		Dropoff_Fix08:=80;
		Weld_Fix08:=81;
		Pickup_Fix08:=82;
		Seal_Fix08:=83;
		Stud_Fix08:=84;
		Sweep_Fix08 := 85;

		Dropoff_Fix09:=90;
		Weld_Fix09:=91;
		Pickup_Fix09:=92;
		Seal_Fix09:=93;
		Stud_Fix09:=94;
		Sweep_Fix09 := 95;

		Dropoff_Fix10:=100;
		Weld_Fix10:=101;
		Pickup_Fix10:=102;
		Seal_Fix10:=103;
		Stud_Fix10:=104;
		Sweep_Fix10 := 105;

		Dropoff_Fix11:=110;
		Weld_Fix11:=111;
		Pickup_Fix11:=112;
		Seal_Fix11:=113;
		Stud_Fix11:=114;
		Sweep_Fix11 := 115;

		Dropoff_Fix12:=120;
		Weld_Fix12:=121;
		Pickup_Fix12:=122;
		Seal_Fix12:=123;
		Stud_Fix12:=124;
		Sweep_Fix15 := 125;

		Dropoff_Fix13:=130;
		Weld_Fix13:=131;
		Pickup_Fix13:=132;
		Seal_Fix13:=133;
		Stud_Fix13:=134;
		Sweep_Fix13 := 135;

		Dropoff_Fix14:=140;
		Weld_Fix14:=141;
		Pickup_Fix14:=142;
		Seal_Fix14:=143;
		Stud_Fix14:=144;
		Sweep_Fix14 := 145;

		Dropoff_Fix15:=150;
		Weld_Fix15:=151;
		Pickup_Fix15:=152;
		Seal_Fix15:=153;
		Stud_Fix15:=154;
		Sweep_Fix15 := 155;

		Dropoff_Fix16:=160;
		Weld_Fix16:=161;
		Pickup_Fix16:=162;
		Seal_Fix16:=163;
		Stud_Fix16:=164;
		Sweep_Fix16 := 165;

		(*Tasks Associated with Entire Work Area*)
		Dropoff_Fix101:=200;
		Weld_Fix101:=201;
		Pickup_Fix101:=202;
		Sweep_Fix101:=203;

		Dropoff_Fix102:=204;
		Weld_Fix102:=205;
		Pickup_Fix102:=206;
		Sweep_Fix102:=207;

		Dropoff_Fix103:=208;
		Weld_Fix103:=209;
		Pickup_Fix103:=210;

		Dropoff_Fix104:=212;
		Weld_Fix104:=213;
		Pickup_Fix104:=214;

		Dropoff_Fix105:=216;
		Weld_Fix105:=217;
		Pickup_Fix105:=218;

		Dropoff_Fix106:=220;
		Weld_Fix106:=221;
		Pickup_Fix106:=222;

		Dropoff_Fix107:=224;
		Weld_Fix107:=225;
		Pickup_Fix107:=226;

		Dropoff_Fix108:=228;
		Weld_Fix108:=229;
		Pickup_Fix108:=230;

		Dropoff_Fix109:=232;
		Weld_Fix109:=233;
		Pickup_Fix109:=234;

		Work_Ped01:= 241;
		Work_Ped02:= 242;
		Work_Ped03:= 243;
		Work_Ped04:= 244;
		Work_Ped05:= 245;
		Work_Ped06:= 246;
		Work_Ped07:= 247;
		Work_Ped08:= 248;
		Work_Ped09:= 249;
		Work_Ped10:= 250;
		Work_Ped11:= 251;
		Work_Ped12:= 252;
		Work_Ped13:= 253;
		Work_Ped14:= 254;
		Work_Ped15:= 255;
		Work_Ped16:= 256;
		Work_Ped17:= 257;
		Work_Ped18:= 258;
		Work_Ped19:= 259;
		Work_Ped20:= 260;
		Work_Ped21:= 261;
		Work_Ped22:= 262;
		Work_Ped23:= 263;
		Work_Ped24:= 264;
		Work_Ped25:= 265;
		Work_Ped26:= 266;
		Work_Ped27:= 267;
		Work_Ped28:= 268;
		Work_Ped29:= 269;
		Work_Ped30:= 270;

		Master_Test:= 351;
		Brake_Test:= 352;
		Tip_Dress:=353;
		Tip_Change_EXT:=354;
		Tip_Change:=355;
		Tracc_Tcp:=356;

		(*Robot Types*)
		MOTO_ERC:=1;
		MOTO_MRC:=2;
		MOTO_XRC:=10;
		MOTO_NX100:=20;
		MOTO_DX100:=30;
		MOTO_DX100_Dual:=31;
		MOTO_DX100_32:=40;

		KUKA_KRC2:=51;

		KUKA_KRC4:=60;
		KUKA_KRC4_SAFEOP:=61;
		KUKA_KRC4_SAFEOP_Small:=62;
		KUKA_KRC4_SafeOP_ATI:=63;
		KUKA_KRC4c_SAFEOP_AGILUS:=64;

		KUKA_KRC4_SAFEOP_TurnTable:=69;

END_PROGRAM

// ---- POUs/Misc/Ped_Stations.TcPOU
(*!!!!!!!!!!!!!!!!!!!!!!!!!!!!!!!!!!!!!!!!!!!!!!!!!!!!!!!!!!!!!!!!!!!!!!!!!!!!!!!!!!!!!!!!!!!!!!!!!!!!!!!!!!!!!!!!!!!!!!!!!!!!!!!!!!!!!!!!!!!!!!!!!!!!!!!!!!
Program Used to group all Ped Type Station Instances
	author: Brent Lekx-Toniolo of Sodecia GTAC
	Feb, 2015
--------------------------------------------------------------------------------------------------------------
REVISION NOTES:
	Date: Feb 2015
	- Original Concept, b.lekx-toniolo

--------------------------------------------------------------------------------------------------------------
*)
PROGRAM Ped_Stations
	VAR_INPUT
		Enable_Prog: BOOL;
	END_VAR

	VAR
	END_VAR

	(*data that needs to be retained in the event of a power cycle*)
	VAR PERSISTENT
	END_VAR

	VAR_OUTPUT
		Prog_Ok: BOOL;
	END_VAR


(*Set Prog_OK to True*)
Prog_OK:= TRUE;

(*Sic Marking*)
(*PED01*)
MAIN.Ped[1]
	(
	(*FB Inputs*)
	Enable_Motion:= MAIN.Control_Power_ON,
	NodeLayout:= Main.ECAT_Master.PedNodeLayout[1],	(*Pass in Assembled Node layout for UI*)
	Input_Node_Count:= 0,							(*Amount of EP1008 blocks on ped*)
	Output_Node_Count:= 0,							(*Amount of EP2028 or 2624 blocks on ped*)
	VB_Node_Count:= 0,								(*Amount of Valve Banks on ped*)
	Option_SwingCylinder:= FALSE, 					(*Enable Swing Cylinder, can be for Ped Item Swing or Tip Dressers (Must be set to TRUE for Tip Dresser)*)
	Option_TipDresser:= FALSE, 						(*Enable TipDresser functionality*)
	Option_TipChanger:= FALSE, 						(*Enable TipChanger functionality*)
	Part_Present_Count:= 0,							(*Enable use of Part Presents. 0-4 max*)
	Prev_EcatNode_Present:= TRUE,					(*Ensure Previous Node Exists to determine Ecat Cable Break of this Devices Input Cable*)
	Mode_Select:= 1, (*2=Manual, 1=Auto*)
	Model_Data:= EOAT04_2_ProductData_Pers.Product_Model_ID,
	Task_Data:= Work_Ped01,
	Dry_Cycle:= GTAC_CONFIG.Dry_Cycle_Enabled,
	Cell_In_Services:= Cell_Services_Prog.Service_Call_ForAllRobots OR In_From_ICxx.Cycle_Hold,
	PrevProcess_Complete:= EOAT04.Part2_In_EOAT AND ((EOAT04_2_ProductData_Pers.Generic_PassFail_Notes[12] = 'Pass') OR (EOAT04_1_ProductData_Pers.Generic_PassFail_Notes[5] = 'Comp')), 		(*Add Interlock here for a previous process that must be completed before starting this Ped process*)
	Blank_Position_Checks:= FALSE,		(*Use this input with caution, used to blank position checking during welding for example*)
	Start_TipDress_Cycle:= FALSE,		(*When TipDress functionality is enable, holding this input high will start the tip dress cycle*)
	Start_TipChange_Cycle:= FALSE,		(*When TipChange functionality is enable, holding this input high will start the tip change cycle*)
	Swing_Adv_REQ:= FALSE,
	Swing_Ret_REQ:= FALSE,
	Tool_at_Home:= TRUE,			(*Conditions for Ped HOME position*)
	Tool_At_Work0:= TRUE,			(*Conditions for Ped WORK position with cylinder*)
	Tool_At_Work1:= FALSE,			(*Conditions for Ped WORK position with cylinder*)
	Work_Robots_Clear:=  (MAIN.R4.Clear_Of_EquipInterf9 AND NOT (MAIN.R4.Task_ID_Ack=Work_Ped01)) OR MAIN.R4.At_Home,
	Work_Robots_WorkingOK:= (MAIN.R4.Task_ID_Ack=Work_Ped01) AND MAIN.R4.Operating,
	Work_Robots_Complete:= MAIN.R4.At_EquipInterf9 AND (MAIN.R4.Task_ID_Ack=Work_Ped01) AND MAIN.R4.Task_Completed,
	Work_Robots_CommonPartInEOAT:= EOAT04.Part2_In_EOAT, 					(*Will set Fix_ID=1*)
	Work_Robots_LHPartInEOAT:= FALSE, 		(*Will set Fix_ID=2*)
	Work_Robots_RHPartInEOAT:= FALSE, 		(*Will set Fix_ID=3*)
	Work_Robots_EOATEmpty:= EOAT04.EOAT_Part2_Empty,
	Part_Present1_REQ:= FALSE,
	Part_Present2_REQ:= FALSE,
	Part_Present3_REQ:= FALSE,
	Part_Present4_REQ:= FALSE,
	Output_Node_UserREQS:= 0, 	(*Allow control of Output Node N50.Q.0 thru.7 (.0 and .1 reserved if TipDress Option is Enabled*)
	(*FB Outputs*)
	Cycle_Time_Out=> ,
	PrevCycle_Time_Out=> ,
	Tool_Call_ForWorkRobots=> , (*Mapped in Robot_Interlock_Map*)
	Robots_Clear_ToProceed=> R1_Data.Proceed_From_Pounce[17],
	Task_ID=> R4_Data.Task_ID[17],
	Fix_ID=> R4_Data.Fix_ID[17],
	Model_ID=> R4_Data.Model_ID[17],
	Work_Complete_Ack=> R4_Data.Complete_Ack[17],
	Repo_Ack=> R4_Data.PeripheralReq_Ack[17]
	);
	(*Map Outputs from Ped01*)
	R4_Data.AuxReq_Ack[17].0:= ((MAIN.R4.Task_ID_Ack=Work_Ped01) AND MAIN.R4.Peripheral_Req.0) AND Out_To_ICxx.SIC01_Complete;


(*Add more peds as required, up to 30 peds*)
	
	(*Move all PedXX data to the Out_To_ICxx Image*)
	Out_to_ICxx.PED[1] :=Main.Ped[1].Discrete_Image;
	Out_to_ICxx.PED[2] :=Main.Ped[2].Discrete_Image;
	Out_to_ICxx.PED[3] :=Main.Ped[3].Discrete_Image;
	Out_to_ICxx.PED[4] :=Main.Ped[4].Discrete_Image;
	Out_to_ICxx.PED[5] :=Main.Ped[5].Discrete_Image;
	Out_to_ICxx.PED[6] :=Main.Ped[6].Discrete_Image;
	Out_to_ICxx.PED[7] :=Main.Ped[7].Discrete_Image;
	Out_to_ICxx.PED[8] :=Main.Ped[8].Discrete_Image;
	Out_to_ICxx.PED[9] :=Main.Ped[9].Discrete_Image;
	Out_to_ICxx.PED[10] :=Main.Ped[10].Discrete_Image;
	Out_to_ICxx.PED[11] :=Main.Ped[11].Discrete_Image;
	Out_to_ICxx.PED[12] :=Main.Ped[12].Discrete_Image;
	Out_to_ICxx.PED[13] :=Main.Ped[13].Discrete_Image;
	Out_to_ICxx.PED[14] :=Main.Ped[14].Discrete_Image;
	Out_to_ICxx.PED[15] :=Main.Ped[15].Discrete_Image;
	Out_to_ICxx.PED[16] :=Main.Ped[16].Discrete_Image;
	Out_to_ICxx.PED[17] :=Main.Ped[17].Discrete_Image;
	Out_to_ICxx.PED[18] :=Main.Ped[18].Discrete_Image;
	Out_to_ICxx.PED[19] :=Main.Ped[19].Discrete_Image;
	Out_to_ICxx.PED[20] :=Main.Ped[20].Discrete_Image;
	Out_to_ICxx.PED[21] :=Main.Ped[21].Discrete_Image;
	Out_to_ICxx.PED[22] :=Main.Ped[22].Discrete_Image;
	Out_to_ICxx.PED[23] :=Main.Ped[23].Discrete_Image;
	Out_to_ICxx.PED[24] :=Main.Ped[24].Discrete_Image;
	Out_to_ICxx.PED[25] :=Main.Ped[25].Discrete_Image;
	Out_to_ICxx.PED[26] :=Main.Ped[26].Discrete_Image;
	Out_to_ICxx.PED[27] :=Main.Ped[27].Discrete_Image;
	Out_to_ICxx.PED[28] :=Main.Ped[28].Discrete_Image;
	Out_to_ICxx.PED[29] :=Main.Ped[29].Discrete_Image;
	Out_to_ICxx.PED[30] :=Main.Ped[30].Discrete_Image;

END_PROGRAM

// ---- POUs/Misc/Ancillary_Equipment.TcPOU
(*!!!!!!!!!!!!!!!!!!!!!!!!!!!!!!!!!!!!!!!!!!!!!!!!!!!!!!!!!!!!!!!!!!!!!!!!!!!!!!!!!!!!!!!!!!!!!!!!!!!!!!!!!!!!!!!!!!!!!!!!!!!!!!!!!!!!!!!!!!!!!!!!!!!!!!!!!!
Program Used to group all Ancillary Equipment (Stud Controller, Sealant Controllers etc)
	author: Brent Lekx-Toniolo of Sodecia GTAC
	March, 2015
--------------------------------------------------------------------------------------------------------------
REVISION NOTES:
	Date: March 2015
	- Original Concept, b.lekx-toniolo

--------------------------------------------------------------------------------------------------------------
*)

PROGRAM Ancillary_Equipment
	VAR_INPUT
		Enable_Prog: BOOL;
	END_VAR

	VAR
		SIC01_Filename: STRING(12); 					(*12 character string that can be sent to the SIC marker to change the program name*)
		SIC01_Variables: ARRAY[1..11] OF STRING[16]; 	(*16 Character string that can be sent to the SIC marker as variables controlled by the PLC.*)
		
		VFD1_OffDelay: TON;
		VFD1_OffDelay2: TON;
		VFD_OnOFF: SR;
		
		VFD2_OffDelay: TON;
		VFD2_OffDelay2: TON;
		VFD2_OnOFF: SR;

		
		Reset_NutOK: INT;
		SIC01_Start_FumeExtractor: BOOL;
		SIC01_Start_OffDelay: TOF;
		SIC01_FumeExtractor_Ready: BOOL;
		SIC01_FumeExtractor_Faulted: BOOL;
		SIC01_FumeExtractor_FilterFault: BOOL;
		SIC01_Variables16: ARRAY[1..8] OF STRING[16]; (* 16 Character string that can be sent to the SIC marker as variables controlled by the PLC. *)
		SIC01_Variables32: ARRAY[9..12] OF STRING[32];
		SIC01_Variables64: ARRAY[13..14] OF STRING[64];
		SIC01_SerialNumberQR: STRING[16];
		SIC01_SerialNumberQR1: STRING[31];
		SIC01_SerialNumberQR2: STRING[16];
		Serial_Number_Transfered_OK: BOOL;
		sYear: STRING[4];
		sTrimYear: STRING[2];
		sDOY: STRING[3];
		sItemNumber: STRING[10];
		wDOY: WORD;
		wYear: WORD;
		wMonth: WORD;
		wDay: WORD;
		weekOfYear: WORD;
		sWeekOfYear: STRING[2];
		sDayOfWeek: STRING[2];
		PartCountINC: R_TRIG;
		Current_Time: DT;
		Current_Time_Unix: UDINT;
		KeepOpenTime: DINT;
		Current_Time_DT: DT;
		Current_Time_DTplus: DT;
		sCurrent_Time_DTplus: STRING[22];
		(*KOT = Keep Open Time*)
		sYear_KOT: STRING[4];
		sTrimYear_KOT: STRING[2];
		sMonth_KOT: STRING[2];
		sDOY_KOT: STRING[2];
		wDOY_KOT: WORD;
		wYear_KOT: WORD;
		wMonth_KOT: WORD;
		wDay_KOT: WORD;
		KeepOpenDate: TIMESTRUCT;
		lint_DOY_KOT: LINT;
		lint_Month_KOT: LINT;
		lint_DOY: LINT;
		sDrawingNumber: String[3];
		(*Keep Open Date Formulation*)
		sKOD_Year_KOT: STRING[4];
		sKOD_TrimYear_KOT: STRING[2];
		sKOD_Month_KOT: STRING[2];
		sKOD_DOY_KOT: STRING[2];
		wKOD_DOY_KOT: WORD;
		wKOD_Year_KOT: WORD;
		wKOD_Month_KOT: WORD;
		wKOD_Day_KOT: WORD;
		sPart_Name : STRING[4];
		Current_Shift: STRING[1];
		DrawingLetter: STRING[255];
		
		SafeGuard01_ADVD: BOOL;
		SafeGuard01_RETD: BOOL;
		
		
END_VAR

	(*data that needs to be retained in the event of a power cycle*)
	VAR PERSISTENT
		ItemNumber: DINT;
		ProductionCount: UINT;
		sProductionCount: STRING[5];
		lint_ProductionCount: LINT;
		DrawingNumberInput: STRING[255];
		PaddedDrawingNumber: STRING[255];
		PaddedDrawingLetter: STRING[255];
		PartChangeNumber: STRING[1];
		DrawingLetterInput: STRING[1];
		FormattedDrawingNumber: STRING[3];
	END_VAR

	VAR_OUTPUT
		Prog_Ok: BOOL;
	END_VAR

	(*Set Prog_OK to True*)
	Prog_OK:= TRUE;

	(*SIC Marking Controller #1*)
	MAIN.SIC01(
        Enable_Motion:= (MAIN.All_SafetyGates_OK AND MAIN.All_Estops_OK),

		Comm_Method:= 2, (*Comm Method 1 is the older method of all string characters, Comm method 2 is the newer method of the data no GSD changes requried between the two modes*)
		FileName_string:= SIC01_FileName,

		LoadFile_bool:= ((MAIN.R4.Task_ID_Ack=Work_PED01) OR MAIN.SIC01.Retry ),
		Start_bool:=  (Main.Ped[1].Enable_Motion AND (MAIN.R4.Task_ID_Ack=Work_Ped01) AND MAIN.R4.Peripheral_Req.0 AND NOT MAIN.SIC01.Retry),

		ResetError_bool:= In_From_ICxx.ControlPower1,
		CompleteReset_bool:= MAIN.PED[1].Work_Robots_Complete,
		Bypass_bool:= In_From_ICxx.SIC01_BypassReq,
		Variables:= SIC01_Variables,

		DpState=> Out_To_ICxx.SIC01_DpState,
		Profinode_OK_bool=> Out_To_ICxx.SIC01_ProfinodeOK,
		SIC_Running_bool=> Out_To_ICxx.SIC01_Running,
		LastDot_bool=> Out_To_ICxx.SIC01_LastDot,
		BackHome_bool=> Out_To_ICxx.SIC01_BackHome,
		Complete_bool=> Out_To_ICxx.SIC01_Complete,
		DataReceived_string=> Out_To_ICxx.SIC01_Reply
		);
		(*Variables to Send to be printed*)
		SIC01_Variables[1]:= FormattedDrawingNumber; 		
		SIC01_Variables[2]:= Current_Shift; 	
		SIC01_Variables[3]:= CONCAT('R',sDayOfWeek); 	
		SIC01_Variables[4]:= CONCAT('R',sWeekOfYear); 
		SIC01_Variables[5]:= CONCAT('R',sTrimYear); 
		SIC01_Variables[6]:= EOAT04_2_ProductData_Pers.Product_Number;
		
		(*Call to Action*)
		DMC_Code_Formation();


		
(*----------------------Motorized Roll Up Doors Controllers-------------------*)

(*New Style Doors with it's own I/O*)
	(*Motorized Roll Up Door #1 Control*)

	MAIN.MD01(
		(*FB Inputs*)
		Enable_Motion:= MAIN.All_Estops_OK AND MAIN.IC01.OP1_LC_Clear,
		CoE_Read_Trigger:= (GTAC_CONFIG.Option_MD_Count>=1) AND Pulse_CoERead,	(*Global Interval of CoE Reads*)
		Ecat_Master_AmsNetID:= MAIN.ECAT_Master.AmsID,
		Prev_EcatNode_Present:= NOT MAIN.IC01.EK1100_NotPresent, (*Ensure Previous Node Exists to determine Ecat Cable Break of this Devices Input Cable*)
        Enable_Latch:= TRUE,
		Fault_Time:= T#3S,
		
		Safety_RST:= MAIN.SAFETY_RESET,
		OPxx_RST:= MAIN.IC01.OP1_Cycle_Start OR MAIN.IC01.OP2_Cycle_Start,

		DoorClose_REQ:= (((Fix01.Door_Close_Req AND FIX01.TurntableB_At_Robot)
						OR (Fix02.Door_Close_Req AND FIX02.TurntableA_At_Robot)) AND MAIN.IC01.OP1_LC_Clear),
		DoorOpen_REQ:= ((Fix01.Door_Open_Req AND FIX01.TurntableB_At_Robot)
						OR (Fix02.Door_Open_Req AND FIX02.TurntableA_At_Robot)),
		DoorStop_REQ:= (*Fix01.Door_Close_Req OR Fix02.Door_Close_Req*)NOT MAIN.IC01.OP1_LC_Clear,

		DoorClosed_Safety_Switches:= MAIN.MD01_N01_I0 AND MAIN.MD01_N01_I1 AND MAIN.MD01_N01_I2 AND MAIN.MD01_N01_I3,		(*Debug Tie in Switch Inputs here*)
		
		(*FB Outputs*)
		DoorClose_CMD=> , 
		DoorOpen_CMD=> ,  
		Door_Closed=>,
		Door_Opened=> ,
		Door_Stopped=>,
		Door_Faulted=>,
		);
		Out_To_ICxx.MD[1].Discrete_Image:= MAIN.MD01.Discrete_Image;
		Out_To_ICxx.MD[1].ECAT_Cable_Breaks:= MAIN.MD01.ECatSlave_Cable_Breaks;
		
		
	MAIN.MD02(
		(*FB Inputs*)
		Enable_Motion:= MAIN.All_Estops_OK AND MAIN.IC02.OP1_LC_Clear,
		Prev_EcatNode_Present:= NOT MAIN.MD01.EP2624_PortB_MissingLink, (*Ensure Previous Node Exists to determine Ecat Cable Break of this Devices Input Cable*)
        Enable_Latch:= TRUE,
		Fault_Time:= T#3S,
		
		Safety_RST:= MAIN.SAFETY_RESET,
		OPxx_RST:= MAIN.IC02.OP1_Cycle_Start OR MAIN.IC02.OP2_Cycle_Start,
		
		DoorClose_REQ:= (((Fix03.Door_Close_Req AND FIX03.TurntableB_At_Robot)
						OR (Fix04.Door_Close_Req AND FIX04.TurntableA_At_Robot)) AND MAIN.IC02.OP1_LC_Clear),
		DoorOpen_REQ:= ((Fix03.Door_Open_Req AND FIX03.TurntableB_At_Robot)
						OR (Fix04.Door_Open_Req AND FIX04.TurntableA_At_Robot)),
		DoorStop_REQ:= (*Fix03.Door_Close_Req OR Fix04.Door_Close_Req*)NOT MAIN.IC02.OP1_LC_Clear,

		DoorClosed_Safety_Switches:= MAIN.MD02_N01_I0 AND MAIN.MD02_N01_I1 AND MAIN.MD02_N01_I2 AND MAIN.MD02_N01_I3,		(*Debug Tie in Switch Inputs here*)

		(*FB Outputs*)
		DoorClose_CMD=> , 
		DoorOpen_CMD=> ,  
		Door_Closed=>,
		Door_Opened=> ,
		Door_Stopped=>,
		Door_Faulted=>,
		);
		Out_To_ICxx.MD[2].Discrete_Image:= MAIN.MD02.Discrete_Image;
		Out_To_ICxx.MD[2].ECAT_Cable_Breaks:= MAIN.MD02.ECatSlave_Cable_Breaks;
		
		
		(*
	(*Internal MD*)	
	MAIN.MD03(
		(*FB Inputs*)
		Enable_Motion:= MAIN.All_Estops_OK AND MAIN.IC01.OP1_LC_Clear,
		Prev_EcatNode_Present:= NOT MAIN.ESW03.EP1908_NotPresent, (*Ensure Previous Node Exists to determine Ecat Cable Break of this Devices Input Cable*)
        Enable_Latch:= TRUE,
		Fault_Time:= T#3S,

		DoorClose_REQ:= (Fix05.Door_Close_Req AND MAIN.IC01.OP1_LC_Clear),
		DoorOpen_REQ:= Fix05.Door_Open_Req,
		DoorStop_REQ:= Fix05.Door_Close_Req,

		DoorClosed_Safety_Switches:= ,		(*Debug Tie in Switch Inputs here*)

		(*FB Outputs*)
		DoorClose_CMD=> , 
		DoorOpen_CMD=> ,  
		Door_Closed=>,
		Door_Opened=> ,
		Door_Stopped=>,
		Door_Faulted=>,
		);
		Out_To_ICxx.MD[3].Discrete_Image:= MAIN.MD03.Discrete_Image;
		Out_To_ICxx.MD[3].ECAT_Cable_Breaks:= MAIN.MD03.ECatSlave_Cable_Breaks;
		
		*)
		
SafeGuard01_ADVD:= MAIN.VertiGuard_N02.I.0 AND MAIN.VertiGuard_N02.I.1;
SafeGuard01_RETD:= MAIN.VertiGuard_N02.I.2 AND MAIN.VertiGuard_N02.I.3;


		
			(*Safety Guard Controller for SafeGate 01*)
	MAIN.VertiGuard_1(
					(*FB Inputs*)
					Enable_FB:= TRUE,
					Enable_Motion:= MAIN.All_Estops_OK (*AND MAIN.IC01.OP1_LC_Clear*),
					Enable_Latch:= TRUE,

					GateOpened_Time:= T#500MS,					(*set this to delay the door open output, set to 500ms if door swtiches are used*)
					GateClosed_Time:= T#500MS,					(*door closed delay*)
					GateOpen_Precharge_Time:= T#0.5S,			(*Door Open Precharge Time*)
					Fault_Time:= T#10S,

					GateClose_REQ:= Fix102.Guard_Close_Req,
					GateOpen_REQ:= Fix102.Guard_Open_Req,

					GateClosed_Switches:= SafeGuard01_ADVD, 
					GateOpened_Switches:= SafeGuard01_RETD, 

					(*FB Outputs*)
					GateClose_CMD=> , (*Mapped in Main*)
					GateOpen_CMD=> ,  (*Mapped in Main*)
					Gate_Closed=> ,
					Gate_Opened=> ,
					Faulted=>
			);
		
(*------------------------------------- Conveyors --------------------------------------*)	
	(*Debug example only*)
		
	(*Conveyor 01*)
	MAIN.Conveyor01(
		Enable_Motion:= MAIN.All_SafetyGates_OK AND MAIN.All_Estops_OK,
		Enable_Start_Latch:= TRUE,				(*Set to True if you want the conveyor to run until the stop signal is activated*)

		Start_Delay_Time:= T#1s,					(*Use this to delay the start of the conveyor signal.Set to T#0s if you dont want to use this.*)
		Stop_Delay_Time:= T#250ms,				(*use this to delay the stop of the conveyor signal. Set to T#0s if you dont want to use this.*)

		Start_Conveyor:= FALSE,					(*Start signal to conveyor*)
		Stop_Conveyor:= FALSE,					(*Stop signal to conveyor*)

		FB_OK=> ,
		Conveyor_On_CMD=>						(*Mapp to output where the conveyor is being turned on and off*)
		);


(*Finished Part Outfeed - Conveyor*)
	MAIN.VFD01(
		Enable_Motion:= MAIN.All_Estops_OK AND MAIN.All_SafetyGates_OK,
		All_Safeties_OK:= MAIN.All_Estops_OK AND MAIN.All_SafetyGates_OK,
		Prev_EcatNode_Present:= (Fix103.N02.InfoData.State = 8), //debug - check proper ecat - rj

		Operating_State_Switch_On:= NOT VFD1_OffDelay.Q AND NOT VFD1_OffDelay2.Q,
		Enable_Voltage:= NOT VFD1_OffDelay.Q AND NOT VFD1_OffDelay2.Q,
		Operating_State_Quick_Stop_Req:= NOT VFD1_OffDelay.Q AND NOT VFD1_OffDelay2.Q,
		Enable_Operation:= NOT VFD1_OffDelay.Q AND NOT VFD1_OffDelay2.Q,
		Fault_Reset:= In_From_ICxx.ControlPower1,
		Halt:= FALSE,

		Requested_Freq:= 50, (*Enter Value Between 0 and 50*)

		FB_OK=> ,
		Operating_State_Ready=> ,
		Operating_State_Switched_On=> ,
		Operating_State_Operation_enabled=> ,
		Operating_State_Fault=> , 
		Voltage_Enabled=> ,
		Operating_State_Quick_Stop=> , 
		Operating_State_Switch_On_Dissabled=> , 
		Error_Class0=> , 
		Halt_Requested=> , 
		Remote=> ,
		Target_Reached=> ,
		Internal_Limit=> ,
		Operating_Mode_Specific=> ,
		X_ERR=> ,
		X_End=> ,
		Ref_OK=> ,
		Discrete_Image=> );
		
		Out_To_ICxx.VFD[1].Discrete_Image:= MAIN.VFD01.Discrete_Image;
		
		(*If sensor is on for 5 seconds, shut off outfeed conveyor*)
		VFD1_OffDelay(
					IN:= Fix102.Part_Present1 AND NOT In_From_ICxx.ControlPower1,
					PT:= T#5s,
					Q=> ,
					ET=> );

		(*If Fixture 105 is in Auto for longer than x time and the sensor on the belt does not come on or the fixture is put into manual,  then stop the outfeed conveyor*)
		VFD1_OffDelay2(
					IN:= ((Fix102.In_Auto AND NOT Fix102.Part_Present3) OR Fix105.In_Manual)
						AND NOT In_From_ICxx.ControlPower1,
					PT:= T#130s,
					Q=> ,
					ET=> );
					
	MAIN.VFD02(
		Enable_Motion:= MAIN.All_Estops_OK AND MAIN.All_SafetyGates_OK,
		All_Safeties_OK:= MAIN.All_Estops_OK AND MAIN.All_SafetyGates_OK,
		Prev_EcatNode_Present:= (Fix104.N02.InfoData.State = 8), //debug - check proper ecat - rj

		Operating_State_Switch_On:= NOT VFD2_OffDelay.Q AND NOT VFD2_OffDelay2.Q,
		Enable_Voltage:= NOT VFD2_OffDelay.Q AND NOT VFD2_OffDelay2.Q,
		Operating_State_Quick_Stop_Req:= NOT VFD2_OffDelay.Q AND NOT VFD2_OffDelay2.Q,
		Enable_Operation:= NOT VFD2_OffDelay.Q AND NOT VFD2_OffDelay2.Q,
		Fault_Reset:= In_From_ICxx.ControlPower1,
		Halt:= FALSE,

		Requested_Freq:= 50, (*Enter Value Between 0 and 50*)

		FB_OK=> ,
		Operating_State_Ready=> ,
		Operating_State_Switched_On=> ,
		Operating_State_Operation_enabled=> ,
		Operating_State_Fault=> , 
		Voltage_Enabled=> ,
		Operating_State_Quick_Stop=> , 
		Operating_State_Switch_On_Dissabled=> , 
		Error_Class0=> , 
		Halt_Requested=> , 
		Remote=> ,
		Target_Reached=> ,
		Internal_Limit=> ,
		Operating_Mode_Specific=> ,
		X_ERR=> ,
		X_End=> ,
		Ref_OK=> ,
		Discrete_Image=> );
		
		Out_To_ICxx.VFD[2].Discrete_Image:= MAIN.VFD02.Discrete_Image;
		
		(*If sensor is on for 5 seconds, shut off outfeed conveyor*)
		VFD2_OffDelay(
					IN:= Fix102.Part_Present1 AND NOT In_From_ICxx.ControlPower1,
					PT:= T#5s,
					Q=> ,
					ET=> );

		(*If Fixture 105 is in Auto for longer than x time and the sensor on the belt does not come on or the fixture is put into manual,  then stop the outfeed conveyor*)
		VFD2_OffDelay2(
					IN:= ((Fix102.In_Auto AND NOT Fix102.Part_Present3) OR Fix105.In_Manual)
						AND NOT In_From_ICxx.ControlPower1,
					PT:= T#130s,
					Q=> ,
					ET=> );

ACTION DMC_Code_Formation:

	(*Formation of the String Variables For The DMC Code/Print Data*)
	(*-------------------------------------------------------*)
	
	(*Production Lifetime Counter*)
	PartCountINC.CLK:= Out_To_ICxx.SIC01_Complete;
	PartCountINC();
	
	IF PartCountINC.Q
		THEN
		ProductionCount:= ProductionCount + 1;
	END_IF

	sItemNumber:= DWORD_TO_STRING(ItemNumber);
	lint_ProductionCount:= DWORD_TO_LINT(ProductionCount);
	sProductionCount:= LINT_TO_DECSTR(lint_ProductionCount,5);
	

	(*-------------------------------------------------------*)
	(*Date Formating*)
	sYear:= WORD_TO_STRING(Main.Local_Time.wYear);			(*Convert Year to String*)
	sTrimYear:= DELETE(STR:=sYear,2,2);						(*Remove first two digits to format year to 'YY'*)
	
	(*Get Day of Year and Convert to String*)
	wDOY:= F_GetDOYOfYearMonthDay(Main.Local_Time.wYear, Main.Local_Time.wMonth, Main.Local_Time.wDay );
	lint_DOY:= WORD_TO_LINT(wDOY);
	sDOY:= LINT_TO_DECSTR(lint_DOY,3);	
	
	(*Get Week of the Year Fucntion*)
	weekOfYear := F_GetWeekOfTheYear(Current_Time);
	sWeekOfYear:= WORD_TO_STRING(weekOfYear);				(*Convert Date/Time to String*)		
	
	(*Convert Day of the week to String*)
	sDayOfWeek:= WORD_TO_STRING(Main.Local_Time.wDayOfWeek);
	
	
	(*-------------------------------------------------------*)
	(*Program to use on Flashed memory of SiC Marker*)
	SIC01_FileName:= '01'; 	
	
	
	(*-------------------------------------------------------*)
	(*Keep-Open Time*)
	(*Keep Open time, 1 day is 86400s, customer requested 30 days = 2592000s*)
	KeepOpenTime:= 30 * 86400;
	Current_Time:= SYSTEMTIME_TO_DT(Main.Local_Time);
	Current_Time_Unix:= DT_TO_UDINT(Current_Time);
	
	(*Model Code Addition to Printed string*)
	IF EOAT02.EOAT_Full THEN 
			sPart_Name := '';
	END_IF
	
	(*Example*)
	IF MAIN.Ped[5].Work_Robots_Complete
		THEN
	Current_Time_DTplus:= UDINT_TO_DT(Current_Time_Unix + KeepOpenTime);
	(*Convert to string to send to SiC Marker*)
	sCurrent_Time_DTplus:= DT_TO_STRING(Current_Time_DTplus);
	
	(*Grab YYMMDD for Keep Open Time*)
	KeepOpenDate:= DT_TO_SYSTEMTIME(Current_Time_DTplus);
	(*Year*)
	sYear_KOT:= WORD_TO_STRING(KeepOpenDate.wYear);			(*Convert Year to String*)
	sTrimYear_KOT:= DELETE(STR:=sYear_KOT,2,2);				
	(*Month*)
	lint_Month_KOT:= WORD_TO_LINT(KeepOpenDate.wMonth);
	sMonth_KOT:= LINT_TO_DECSTR(lint_Month_KOT,2);
	(*Day*)
	lint_DOY_KOT:= WORD_TO_LINT(KeepOpenDate.wDay);
	sDOY_KOT:= LINT_TO_DECSTR(lint_DOY_KOT,2);
	
	END_IF
	
	
	(*-------------------------------------------------------*)
	(*User input - Drawing Number*)
	F_FormatArgToStr(
	bSign:= FALSE, 
	bBlank:= FALSE, 
	bNull:= TRUE, 
	bHash:= FALSE, 
	bLAlign:= FALSE, 
	bWidth:= FALSE, 
	iWidth:= 3, 
	iPrecision:= 3, 
	eFmtType:= TYPEFIELD_S, 
	arg:= F_STRING(DrawingNumberInput), 
	sOut:=  PaddedDrawingNumber);
	
	FormattedDrawingNumber:= F_ToUCase(PaddedDrawingNumber);
	
	(*-------------------------------------------------------*)
	(*User input - Part Change Letter*)
	F_FormatArgToStr(
	bSign:= FALSE, 
	bBlank:= FALSE, 
	bNull:= TRUE, 
	bHash:= FALSE, 
	bLAlign:= FALSE, 
	bWidth:= FALSE, 
	iWidth:= 0, 
	iPrecision:= 1, 
	eFmtType:= TYPEFIELD_S, 
	arg:= F_STRING(DrawingLetter), 
	sOut:=  PaddedDrawingLetter);
	
	DrawingLetterInput:= F_ToUCase(PaddedDrawingLetter); (*Force Upper Case - just in case*)
	
	
	(*-------------------------------------------------------*)
	(*Shift Letter*)
	Current_Shift:= Fix01.Production_Report.Shift_Letter;
END_ACTION

END_PROGRAM

// ---- POUs/FBs/FB_Clamp_Status.TcPOU
(*FB for replacement of typical clamp fault checking code":
	Original Author(s): Brent Lekx-Toniolo of Toniolo Research & Development Inc.; 
	August 2010; version 3.0

------------------------------------------------------------------------------------------
REVISION NOTES:
	Version 20170608
		-  Added disable fault input, b.lekx-toniolo / j.underhill

------------------------------------------------------------------------------------------
*)
FUNCTION_BLOCK FB_Clamp_Status
	VAR_INPUT
		Enable_FB: BOOL;
		Home_Sensor: BOOL;
		Work_Sensor: BOOL;
		Home_Solenoid: BOOL;
		Work_Solenoid: BOOL;
		Home_Delay: TIME;
		Work_Delay: TIME;
		Fault_Delay: TIME;
		Disable_Fault: BOOL;
	END_VAR

	VAR
		At_Home: BOOL;
		At_Work: BOOL;
		Home_Delay_TMR: TON;
		Work_Delay_TMR: TON;
		Sensor_FLT_TMR: TON;
		GoingHome_FLT_TMR: TON;
		GoingWork_FLT_TMR: TON;
	END_VAR

	VAR_OUTPUT
		FB_OK: BOOL;
		In_Home_Position: BOOL;
		In_Work_Position: BOOL;
		Faulted: BOOL;
		Sensor_Fault: BOOL;
		GoingToHome_Fault: BOOL;
		GoingToWork_Fault: BOOL;
	END_VAR

	(*Set FB_OK to True*)
	FB_OK:= TRUE;
(*$$$$$$$$$$$$$$$$$$$$$$$$$$$$$$$$$$ Internal Code $$$$$$$$$$$$$$$$$$$$$$$$$$$$$$$$$$$$$$$$$$$$$$$*)
	(*Develop Home Position*)
	At_Home:=Home_Sensor AND NOT Work_Sensor;

	(*Develop Work Position*)
	At_Work:=Work_Sensor AND NOT Home_Sensor;

	(*Delay Home Position Output*)
	Home_Delay_TMR.PT:= Home_Delay;
	Home_Delay_TMR.IN:=At_Home;
	Home_Delay_TMR();
	In_Home_Position:=Home_Delay_TMR.Q;

	(*Delay Work Position Output*)
	Work_Delay_TMR.PT:= Work_Delay;
	Work_Delay_TMR.IN:=At_Work;
	Work_Delay_TMR();
	In_Work_Position:=Work_Delay_TMR.Q;

(*$$$$$$$$$$$$$$$$$$$$$$$$$$$$$$$$$$$$$$$$ Fault Code $$$$$$$$$$$$$$$$$$$$$$$$$$$$$$$$$$$$$$$$$$$$$$$$*)
	(*Sensor Fault*)
	Sensor_FLT_TMR.PT:=Fault_Delay;
	Sensor_FLT_TMR.IN:=(NOT At_Home AND NOT At_Work) OR (At_Work AND At_Home);
	Sensor_FLT_TMR();
	Sensor_Fault:=Sensor_FLT_TMR.Q;

	(*Going Home Fault*)
	GoingHome_FLT_TMR.PT:=Fault_Delay;
	GoingHome_FLT_TMR.IN:=Home_Solenoid AND NOT At_Home AND NOT Sensor_Fault;
	GoingHome_FLT_TMR();
	GoingToHome_Fault:=GoingHome_FLT_TMR.Q;

	(*Going Home Fault*)
	GoingWork_FLT_TMR.PT:=Fault_Delay;
	GoingWork_FLT_TMR.IN:=Work_Solenoid AND NOT At_Work AND NOT Sensor_Fault;
	GoingWork_FLT_TMR();
	GoingToWork_Fault:=GoingWork_FLT_TMR.Q;

	(*Develop Fault Output*)
	Faulted:= NOT Disable_Fault AND (Sensor_Fault OR GoingToHome_Fault OR GoingToWork_Fault);

END_FUNCTION_BLOCK

// ---- POUs/FBs/FB_ENET_Com20131205.TcPOU
FUNCTION_BLOCK FB_ENET_Com20131205

VAR_INPUT

	LocalNetID:						STRING(19);			(*AMS Net ID of PLC*)

	RemotePort:						UDINT;				(*Port on remote device*)
	RemoteIPAddress:				STRING(15);			(*IP Address of Remote Device*)

	SendData:						STRING;

	Connect:							BOOL;				(*Opens the Connection to the Specified device*)
	Send:							BOOL;				(*Sends the data to the Specified device*)



END_VAR
VAR_OUTPUT

	ConnectionError:					BOOL;
	ConnectionErrorID:				UDINT;
	ConnectionState:					E_SocketConnectionState;

	ReceiveData:						STRING;

END_VAR
VAR
	Pulse:							FB_Pulse_Generator;
	Pulse_100ms:						BOOL;


	ClientServerConnection: 			FB_ClientServerConnection;
	SocketSend:						FB_SocketSend;
	SocketReceive:					FB_SocketReceive;

	SocketHandle: 					T_HSocket;

	Received:						STRING;

	CommandLength:					INT;				(*String Length of Command being sent*)
	ReceiveLength:					UDINT;			(*String Length of Received Data*)
	RecLengthINT:					INT;

	pSrc: 							POINTER TO STRING;
	pDest: 							POINTER TO STRING;


END_VAR

pSrc := ADR(SendData);								(*Point to address of the data to be sent*)
pDest := ADR(Received);								(*Point to address of received date*)

CommandLength:= LEN(SendData);
RecLengthINT:= UDINT_TO_INT(ReceiveLength);
ReceiveData:= LEFT(Received, RecLengthINT);

Pulse(On_Time:=T#100ms , Off_Time:= T#100ms, Wave=>Pulse_100ms );



(*---------------------------------------------------------FB Instances------------------------------------------------------*)


(*Opens the socket to the device we are connecting to*)
ClientServerConnection(
	sSrvNetID:= LocalNetID,
	nMode:=0 OR CONNECT_MODE_ENABLEDBG,
	sRemoteHost:=RemoteIPAddress,
	nRemotePort:=RemotePort,
	bEnable:=Connect,
	tReconnect:=T#30s,
	bBusy=> ,
	bError=> ConnectionError,
	nErrId=> ConnectionErrorID,
	hSocket=>SocketHandle,
	eState=> ConnectionState);


(*Send Data to the open handle specified*)
SocketSend(
	sSrvNetId:= LocalNetID,
	hSocket:= SocketHandle,
	cbLen:= CommandLength,
	pSrc:= pSrc,
	bExecute:= Send,
	tTimeout:= T#20s,
	bBusy=> ,
	bError=> ,
	nErrId=> );

(*Receive Data from the open handle specified*)
SocketReceive(
	sSrvNetId:= LocalNetID,
	hSocket:= SocketHandle,
	cbLen:= 50,
	pDest:= pDest,
	bExecute:= Pulse_100ms AND Connect,
	tTimeout:= T#20s,
	bBusy=> ,
	bError=> ,
	nErrId=> ,
	nRecBytes=>ReceiveLength);

END_FUNCTION_BLOCK

// ---- POUs/FBs/FB_GTAC_EOAT_20170704.TcPOU
(*FB for use with Robot EOATs

	Original Author(s): Brent Lekx-Toniolo of Sodecia GTAC.; 
------------------------------------------------------------------------------------------
REVISION NOTES:
	Version 20151105
		- intial concept, b.lekx-toniolo
	Version 20170507
		- made the FB more awesomer, b.lekx-toniolo
	Version 20170704
		- made the FB even more awesomer with valve changes, j.vandongen
		- added in Part_In_EOAT, removed from robot control, j.vandongen
------------------------------------------------------------------------------------------
*)



FUNCTION_BLOCK FB_GTAC_EOAT_20170704

VAR_INPUT
(*General Inputs*)
	Enable_FB: BOOL;
	Enable_Motion: BOOL;
	Dry_Cycle: BOOL;


(*Node Counts and configuration data*)
	Input_Node_Count: UDINT;
	VB_Node_Count: UDINT;
	Part_Present_Count: UDINT;
	Clamp_Count: UDINT;

	All_Sensors_Off_Grp1: BOOL;
	All_Sensors_On_Grp1: BOOL;
	All_Sensors_Off_Grp2: BOOL;
	All_Sensors_On_Grp2: BOOL;
	All_Sensors_Off_Grp3: BOOL;
	All_Sensors_On_Grp3: BOOL;
	All_Sensors_Off_Grp4: BOOL;
	All_Sensors_On_Grp4: BOOL;
	All_Sensors_Off_Grp5: BOOL;
	All_Sensors_On_Grp5: BOOL;
	All_Sensors_Off_Grp6: BOOL;
	All_Sensors_On_Grp6: BOOL;
	All_Sensors_Off_Grp7: BOOL;
	All_Sensors_On_Grp7: BOOL;
	All_Sensors_Off_Grp8: BOOL;
	All_Sensors_On_Grp8: BOOL;

	LH_Part_In_EOAT_Grp: BOOL;
	LH_EOAT_Empty_Grp: BOOL;
	RH_Part_In_EOAT_Grp: BOOL;
	RH_EOAT_Empty_Grp: BOOL;
	Part_In_EOAT_Grp: BOOL;
	EOAT_Empty_Grp: BOOL;

	Tool_At_Home_Grp1: BOOL;
	Tool_At_Work_Grp1: BOOL;
	Tool_At_Home_Grp2: BOOL;
	Tool_At_Work_Grp2: BOOL;
	Tool_At_Home_Grp3: BOOL;
	Tool_At_Work_Grp3: BOOL;
	Tool_At_Home_Grp4: BOOL;
	Tool_At_Work_Grp4: BOOL;
	Tool_At_Home_Grp5: BOOL;
	Tool_At_Work_Grp5: BOOL;
	Tool_At_Home_Grp6: BOOL;
	Tool_At_Work_Grp6: BOOL;
	Tool_At_Home_Grp7: BOOL;
	Tool_At_Work_Grp7: BOOL;
	Tool_At_Home_Grp8: BOOL;
	Tool_At_Work_Grp8: BOOL;

(*Clamp and PP Mapping*)
	MAP_Clamp1_HomeSens: BOOL;
	MAP_Clamp1_WorkSens: BOOL;
	MAP_Clamp1_HomeReqd: BOOL;
	MAP_Clamp1_WorkReqd: BOOL;
	MAP_Clamp2_HomeSens: BOOL;
	MAP_Clamp2_WorkSens: BOOL;
	MAP_Clamp2_HomeReqd: BOOL;
	MAP_Clamp2_WorkReqd: BOOL;
	MAP_Clamp3_HomeSens: BOOL;
	MAP_Clamp3_WorkSens: BOOL;
	MAP_Clamp3_HomeReqd: BOOL;
	MAP_Clamp3_WorkReqd: BOOL;
	MAP_Clamp4_HomeSens: BOOL;
	MAP_Clamp4_WorkSens: BOOL;
	MAP_Clamp4_HomeReqd: BOOL;
	MAP_Clamp4_WorkReqd: BOOL;
	MAP_Clamp5_HomeSens: BOOL;
	MAP_Clamp5_WorkSens: BOOL;
	MAP_Clamp5_HomeReqd: BOOL;
	MAP_Clamp5_WorkReqd: BOOL;
	MAP_Clamp6_HomeSens: BOOL;
	MAP_Clamp6_WorkSens: BOOL;
	MAP_Clamp6_HomeReqd: BOOL;
	MAP_Clamp6_WorkReqd: BOOL;
	MAP_Clamp7_HomeSens: BOOL;
	MAP_Clamp7_WorkSens: BOOL;
	MAP_Clamp7_HomeReqd: BOOL;
	MAP_Clamp7_WorkReqd: BOOL;
	MAP_Clamp8_HomeSens: BOOL;
	MAP_Clamp8_WorkSens: BOOL;
	MAP_Clamp8_HomeReqd: BOOL;
	MAP_Clamp8_WorkReqd: BOOL;
	MAP_Clamp9_HomeSens: BOOL;
	MAP_Clamp9_WorkSens: BOOL;
	MAP_Clamp9_HomeReqd: BOOL;
	MAP_Clamp9_WorkReqd: BOOL;
	MAP_Clamp10_HomeSens: BOOL;
	MAP_Clamp10_WorkSens: BOOL;
	MAP_Clamp10_HomeReqd: BOOL;
	MAP_Clamp10_WorkReqd: BOOL;
	MAP_Clamp11_HomeSens: BOOL;
	MAP_Clamp11_WorkSens: BOOL;
	MAP_Clamp11_HomeReqd: BOOL;
	MAP_Clamp11_WorkReqd: BOOL;
	MAP_Clamp12_HomeSens: BOOL;
	MAP_Clamp12_WorkSens: BOOL;
	MAP_Clamp12_HomeReqd: BOOL;
	MAP_Clamp12_WorkReqd: BOOL;
	MAP_Clamp13_HomeSens: BOOL;
	MAP_Clamp13_WorkSens: BOOL;
	MAP_Clamp13_HomeReqd: BOOL;
	MAP_Clamp13_WorkReqd: BOOL;
	MAP_Clamp14_HomeSens: BOOL;
	MAP_Clamp14_WorkSens: BOOL;
	MAP_Clamp14_HomeReqd: BOOL;
	MAP_Clamp14_WorkReqd: BOOL;
	MAP_Clamp15_HomeSens: BOOL;
	MAP_Clamp15_WorkSens: BOOL;
	MAP_Clamp15_HomeReqd: BOOL;
	MAP_Clamp15_WorkReqd: BOOL;
	MAP_Clamp16_HomeSens: BOOL;
	MAP_Clamp16_WorkSens: BOOL;
	MAP_Clamp16_HomeReqd: BOOL;
	MAP_Clamp16_WorkReqd: BOOL;
	MAP_Clamp17_HomeSens: BOOL;
	MAP_Clamp17_WorkSens: BOOL;
	MAP_Clamp17_HomeReqd: BOOL;
	MAP_Clamp17_WorkReqd: BOOL;
	MAP_Clamp18_HomeSens: BOOL;
	MAP_Clamp18_WorkSens: BOOL;
	MAP_Clamp18_HomeReqd: BOOL;
	MAP_Clamp18_WorkReqd: BOOL;
	MAP_Clamp19_HomeSens: BOOL;
	MAP_Clamp19_WorkSens: BOOL;
	MAP_Clamp19_HomeReqd: BOOL;
	MAP_Clamp19_WorkReqd: BOOL;
	MAP_Clamp20_HomeSens: BOOL;
	MAP_Clamp20_WorkSens: BOOL;
	MAP_Clamp20_HomeReqd: BOOL;
	MAP_Clamp20_WorkReqd: BOOL;

	MAP_PP1_Sens: BOOL;
	MAP_PP1_ReqdOn: BOOL;
	MAP_PP1_ReqdOff: BOOL;
	MAP_PP2_Sens: BOOL;
	MAP_PP2_ReqdOn: BOOL;
	MAP_PP2_ReqdOff: BOOL;
	MAP_PP3_Sens: BOOL;
	MAP_PP3_ReqdOn: BOOL;
	MAP_PP3_ReqdOff: BOOL;
	MAP_PP4_Sens: BOOL;
	MAP_PP4_ReqdOn: BOOL;
	MAP_PP4_ReqdOff: BOOL;
	MAP_PP5_Sens: BOOL;
	MAP_PP5_ReqdOn: BOOL;
	MAP_PP5_ReqdOff: BOOL;
	MAP_PP6_Sens: BOOL;
	MAP_PP6_ReqdOn: BOOL;
	MAP_PP6_ReqdOff: BOOL;
	MAP_PP7_Sens: BOOL;
	MAP_PP7_ReqdOn: BOOL;
	MAP_PP7_ReqdOff: BOOL;
	MAP_PP8_Sens: BOOL;
	MAP_PP8_ReqdOn: BOOL;
	MAP_PP8_ReqdOff: BOOL;



(*CMDs (commands)*)
	CMD_CheckAllSensors_OFF: BOOL;
	CMD_CheckAllSensors_ON: BOOL;
	CMD_CheckSensorsOFF_Grp1: BOOL;
	CMD_CheckSensorsON_Grp1: BOOL;
	CMD_CheckSensorsOFF_Grp2: BOOL;
	CMD_CheckSensorsON_Grp2: BOOL;
	CMD_CheckSensorsOFF_Grp3: BOOL;
	CMD_CheckSensorsON_Grp3: BOOL;
	CMD_CheckSensorsOFF_Grp4: BOOL;
	CMD_CheckSensorsON_Grp4: BOOL;
	CMD_CheckSensorsOFF_Grp5: BOOL;
	CMD_CheckSensorsON_Grp5: BOOL;
	CMD_CheckSensorsOFF_Grp6: BOOL;
	CMD_CheckSensorsON_Grp6: BOOL;
	CMD_CheckSensorsOFF_Grp7: BOOL;
	CMD_CheckSensorsON_Grp7: BOOL;
	CMD_CheckSensorsOFF_Grp8: BOOL;
	CMD_CheckSensorsON_Grp8: BOOL;

	CMD_Tool_To_WORK: BOOL;
	CMD_Tool_To_HOME: BOOL;
	CMD_ClampsToWORK_Grp1: BOOL;
	CMD_ClampsToHOME_Grp1: BOOL;
	CMD_ClampsToWORK_Grp2: BOOL;
	CMD_ClampsToHOME_Grp2: BOOL;
	CMD_ClampsToWORK_Grp3: BOOL;
	CMD_ClampsToHOME_Grp3: BOOL;
	CMD_ClampsToWORK_Grp4: BOOL;
	CMD_ClampsToHOME_Grp4: BOOL;
	CMD_ClampsToWORK_Grp5: BOOL;
	CMD_ClampsToHOME_Grp5: BOOL;
	CMD_ClampsToWORK_Grp6: BOOL;
	CMD_ClampsToHOME_Grp6: BOOL;
	CMD_ClampsToWORK_Grp7: BOOL;
	CMD_ClampsToHOME_Grp7: BOOL;
	CMD_ClampsToWORK_Grp8: BOOL;
	CMD_ClampsToHOME_Grp8: BOOL;

END_VAR

VAR
(*Hardware Related Data Types*)
			(*Develop "Beckhoff Nodes"*)
			N01 AT %I*: udt_EP1008_002_v2;
			N02 AT %I*: udt_EP1008_002_v2;
			N03 AT %I*: udt_EP1008_002_v2;
			N04 AT %I*: udt_EP1008_002_v2;
			N05 AT %I*: udt_EP1008_002_v2;
			N06 AT %I*: udt_EP1008_002_v2;
			N07 AT %I*: udt_EP1008_002_v2;
			N08 AT %I*: udt_EP1008_002_v2;
			N09 AT %I*: udt_EP1008_002_v2;
			N100 AT %Q*: udt_SMC_EX260_ValveBank;
			N100_STAT AT %I*:udt_SMC_EX260_Stat;

(* Nodes States*)
	DiscreteNode_OK: BOOL;
(* Cable Break States*)
	ECatSlave_Cable_Breaks: UDINT;

(*Standard Internal Variables*)
		(*Generic Sensor Variables*)
		All_Sensors_On: UINT;
		All_Sensors_Off: UINT;
		(*Generic Position Variables*)
		Tool_At_Home: UINT;
		Tool_At_Work: UINT;
		(*General Internals*)
		CLFaulted: UDINT;
		PPFaulted: UDINT;

(*Non-Standard Variables*)

		(*FB Instances*)
		Clamp1FB: FB_Clamp_Status;
		Clamp2FB: FB_Clamp_Status;
		Clamp3FB: FB_Clamp_Status;
		Clamp4FB: FB_Clamp_Status;
		Clamp5FB: FB_Clamp_Status;
		Clamp6FB: FB_Clamp_Status;
		Clamp7FB: FB_Clamp_Status;
		Clamp8FB: FB_Clamp_Status;
		Clamp9FB: FB_Clamp_Status;
		Clamp10FB: FB_Clamp_Status;
		Clamp11FB: FB_Clamp_Status;
		Clamp12FB: FB_Clamp_Status;
		Clamp13FB: FB_Clamp_Status;
		Clamp14FB: FB_Clamp_Status;
		Clamp15FB: FB_Clamp_Status;
		Clamp16FB: FB_Clamp_Status;
		Clamp17FB: FB_Clamp_Status;
		Clamp18FB: FB_Clamp_Status;
		Clamp19FB: FB_Clamp_Status;
		Clamp20FB: FB_Clamp_Status;
		Part_Present1FB: FB_PP_Sensor;
		Part_Present2FB: FB_PP_Sensor;
		Part_Present3FB: FB_PP_Sensor;
		Part_Present4FB: FB_PP_Sensor;
		Part_Present5FB: FB_PP_Sensor;
		Part_Present6FB: FB_PP_Sensor;
		Part_Present7FB: FB_PP_Sensor;
		Part_Present8FB: FB_PP_Sensor;
		Tape_Present1FB: FB_PP_Sensor;
		(*Valve FBs*)
		Valve1FB: FB_GTAC_Valve_20170704;
		Valve2FB: FB_GTAC_Valve_20170704;
		Valve3FB: FB_GTAC_Valve_20170704;
		Valve4FB: FB_GTAC_Valve_20170704;
		Valve5FB: FB_GTAC_Valve_20170704;
		Valve6FB: FB_GTAC_Valve_20170704;
		Valve7FB: FB_GTAC_Valve_20170704;
		Valve8FB: FB_GTAC_Valve_20170704;

		(*Tool Positions*)
			Clamp1WORK: BOOL;
			Clamp1HOME: BOOL;
			Clamp2WORK: BOOL;
			Clamp2HOME: BOOL;
			Clamp3WORK: BOOL;
			Clamp3HOME: BOOL;
			Clamp4WORK: BOOL;
			Clamp4HOME: BOOL;
			Clamp5WORK: BOOL;
			Clamp5HOME: BOOL;
			Clamp6WORK: BOOL;
			Clamp6HOME: BOOL;
			Clamp7WORK: BOOL;
			Clamp7HOME: BOOL;
			Clamp8WORK: BOOL;
			Clamp8HOME: BOOL;
			Clamp9WORK: BOOL;
			Clamp9HOME: BOOL;
			Clamp10WORK: BOOL;
			Clamp10HOME: BOOL;
			Clamp11WORK: BOOL;
			Clamp11HOME: BOOL;
			Clamp12WORK: BOOL;
			Clamp12HOME: BOOL;
			Clamp13WORK: BOOL;
			Clamp13HOME: BOOL;
			Clamp14WORK: BOOL;
			Clamp14HOME: BOOL;
			Clamp15WORK: BOOL;
			Clamp15HOME: BOOL;
			Clamp16WORK: BOOL;
			Clamp16HOME: BOOL;
			Clamp17WORK: BOOL;
			Clamp17HOME: BOOL;
			Clamp18WORK: BOOL;
			Clamp18HOME: BOOL;
			Clamp19WORK: BOOL;
			Clamp19HOME: BOOL;
			Clamp20WORK: BOOL;
			Clamp20HOME: BOOL;
		(*Part Present Sensors*)
			(*Main Body Present*)
			Part_Present1: BOOL;
			Part_Present2: BOOL;
			Part_Present3: BOOL;
			Part_Present4: BOOL;
			Part_Present5: BOOL;
			Part_Present6: BOOL;
			Part_Present7: BOOL;
			Part_Present8: BOOL;



END_VAR

VAR_OUTPUT

		FB_OK: BOOL;
		Discrete_Image: udt_EOATxx_Image_20170607;

		CLFaults1:UDINT;
		CLFaults2:UDINT;
		CLFaults3:UDINT;
		CLFaults4:UDINT;
		PPFaults: UDINT;

		LH_Part_In_EOAT:BOOL;
		RH_Part_In_EOAT:BOOL;
		Part_In_EOAT:BOOL;

(*ACKS*)
	ACK_AllSensors_OFF: BOOL;
	ACK_AllSensors_ON: BOOL;
	ACK_SensorsOFF_Grp1: BOOL;
	ACK_SensorsON_Grp1: BOOL;
	ACK_SensorsOFF_Grp2: BOOL;
	ACK_SensorsON_Grp2: BOOL;
	ACK_SensorsOFF_Grp3: BOOL;
	ACK_SensorsON_Grp3: BOOL;
	ACK_SensorsOFF_Grp4: BOOL;
	ACK_SensorsON_Grp4: BOOL;
	ACK_SensorsOFF_Grp5: BOOL;
	ACK_SensorsON_Grp5: BOOL;
	ACK_SensorsOFF_Grp6: BOOL;
	ACK_SensorsON_Grp6: BOOL;
	ACK_SensorsOFF_Grp7: BOOL;
	ACK_SensorsON_Grp7: BOOL;
	ACK_SensorsOFF_Grp8: BOOL;
	ACK_SensorsON_Grp8: BOOL;

	ACK_Tool_At_WORK: BOOL;
	ACK_Tool_At_HOME: BOOL;
	ACK_ClampsAtWORK_Grp1: BOOL;
	ACK_ClampsAtHOME_Grp1: BOOL;
	ACK_ClampsAtWORK_Grp2: BOOL;
	ACK_ClampsAtHOME_Grp2: BOOL;
	ACK_ClampsAtWORK_Grp3: BOOL;
	ACK_ClampsAtHOME_Grp3: BOOL;
	ACK_ClampsAtWORK_Grp4: BOOL;
	ACK_ClampsAtHOME_Grp4: BOOL;
	ACK_ClampsAtWORK_Grp5: BOOL;
	ACK_ClampsAtHOME_Grp5: BOOL;
	ACK_ClampsAtWORK_Grp6: BOOL;
	ACK_ClampsAtHOME_Grp6: BOOL;
	ACK_ClampsAtWORK_Grp7: BOOL;
	ACK_ClampsAtHOME_Grp7: BOOL;
	ACK_ClampsAtWORK_Grp8: BOOL;
	ACK_ClampsAtHOME_Grp8: BOOL;

END_VAR

	(*Set FB_OK to True*)
	FB_OK:= TRUE;

(*$$$$$$$$$$$$$$$$$$$$$$$$$$$$$$$$$$$$$$$$$$$$$$$$Gather Status Of Hardware $$$$$$$$$$$$$$$$$$$$$$$$$$$$$$$$$$$$$$$$$$$$$$$$$$$$*)
	(*Discrete I/O Nodes*)

	IF N01.InfoData.State=8
		AND (N02.InfoData.State=8 OR (Input_Node_Count<2))
		AND (N03.InfoData.State=8 OR (Input_Node_Count<3))
		AND (N04.InfoData.State=8 OR (Input_Node_Count<4))
		AND (N05.InfoData.State=8 OR (Input_Node_Count<5))
		AND (N06.InfoData.State=8 OR (Input_Node_Count<6))
		AND (N07.InfoData.State=8 OR (Input_Node_Count<7))
		AND (N08.InfoData.State=8 OR (Input_Node_Count<8))
		AND (N09.InfoData.State=8 OR (Input_Node_Count<9))
		AND N100_STAT.InfoData.State=8

		THEN
			DiscreteNode_OK:=TRUE;

	ELSE
			DiscreteNode_OK:=FALSE;

	END_IF;

	(*Cable Break Detection*)
	ECatSlave_Cable_Breaks:= FUN_GTAC_EcatSlaveConnState
							(N100_STAT.InfoData.State,
							N01.InfoData.State ,
							N02.InfoData.State,
							N03.InfoData.State,
							N04.InfoData.State,
							N05.InfoData.State,
							N06.InfoData.State,
							N07.InfoData.State,
							N08.InfoData.State,
							N09.InfoData.State,
							0,0,0,0,0,0,0,0,0,0,0,0,0,0,0,0,0,0,0,0); (*Function Returns Flags to warn of possible cable break*)
(*$$$$$$$$$$$$$$$$$$$$$$$$$$$$$$$$$$$$$$$$$$$$$ Gather Safety Inputs $$$$$$$$$$$$$$$$$$$$$$$$$$$$$$$$$$$$$$$$$$$$$$$$$$$$$$$$$*)


(*$$$$$$$$$$$$$$$$$$$$$$$$$$$$$$$$$$$$$$$$$$$$$ Gather Standard Inputs $$$$$$$$$$$$$$$$$$$$$$$$$$$$$$$$$$$$$$$$$$$$$$$$$$$$$$$$$*)

(*----------------------------------------------------------------------- Gather Clamp Sensor Inputs -----------------------------------------------------*)
(*Clamp/Cylinder Inputs*)
		(*Clamp1*)
		Clamp1FB(
			(*All sensor input mapping and solenoid mapping is done external to FB by end deployment*)
			Home_Sensor:= MAP_Clamp1_HomeSens,
			Work_Sensor:= MAP_Clamp1_WorkSens,
			Home_Solenoid:= Enable_Motion AND (CMD_Tool_To_HOME OR MAP_Clamp1_HomeReqd),
			Work_Solenoid:= Enable_Motion AND (CMD_Tool_To_WORK OR MAP_Clamp1_WorkReqd),
			Home_Delay:= T#0.1s,
			Work_Delay:= T#0.1s ,
			Fault_Delay:= T#3s ,
			In_Home_Position=> Clamp1HOME,
			In_Work_Position=> Clamp1WORK,
			);
			CLFaults1.1:= Clamp1FB.Faulted AND Clamp_Count>=1; 		(*Interlock Clamp Fault with Clamp Count Configuration Data*)

		(*Clamp2*)
		Clamp2FB(
			(*All sensor input mapping and solenoid mapping is done external to FB by end deployment*)
			Home_Sensor:= MAP_Clamp2_HomeSens,
			Work_Sensor:= MAP_Clamp2_WorkSens,
			Home_Solenoid:= Enable_Motion AND (CMD_Tool_To_HOME OR MAP_Clamp2_HomeReqd),
			Work_Solenoid:= Enable_Motion AND (CMD_Tool_To_WORK OR MAP_Clamp2_WorkReqd),
			Home_Delay:= T#0.1s,
			Work_Delay:= T#0.1s ,
			Fault_Delay:= T#3s ,
			In_Home_Position=> Clamp2HOME,
			In_Work_Position=> Clamp2WORK,
			);
			CLFaults1.2:= Clamp2FB.Faulted AND Clamp_Count>=2; 		(*Interlock Clamp Fault with Clamp Count Configuration Data*)
		(*Clamp3*)
		Clamp3FB(
			(*All sensor input mapping and solenoid mapping is done external to FB by end deployment*)
			Home_Sensor:= MAP_Clamp3_HomeSens,
			Work_Sensor:= MAP_Clamp3_WorkSens,
			Home_Solenoid:= Enable_Motion AND (CMD_Tool_To_HOME OR MAP_Clamp3_HomeReqd),
			Work_Solenoid:= Enable_Motion AND (CMD_Tool_To_WORK OR MAP_Clamp3_WorkReqd),
			Home_Delay:= T#0.1s,
			Work_Delay:= T#0.1s ,
			Fault_Delay:= T#3s ,
			In_Home_Position=> Clamp3HOME,
			In_Work_Position=> Clamp3WORK,
			);
			CLFaults1.3:= Clamp3FB.Faulted AND Clamp_Count>=3; 		(*Interlock Clamp Fault with Clamp Count Configuration Data*)
		(*Clamp4*)
		Clamp4FB(
			(*All sensor input mapping and solenoid mapping is done external to FB by end deployment*)
			Home_Sensor:= MAP_Clamp4_HomeSens,
			Work_Sensor:= MAP_Clamp4_WorkSens,
			Home_Solenoid:= Enable_Motion AND (CMD_Tool_To_HOME OR MAP_Clamp4_HomeReqd),
			Work_Solenoid:= Enable_Motion AND (CMD_Tool_To_WORK OR MAP_Clamp4_WorkReqd),
			Home_Delay:= T#0.1s,
			Work_Delay:= T#0.1s ,
			Fault_Delay:= T#3s ,
			In_Home_Position=> Clamp4HOME,
			In_Work_Position=> Clamp4WORK,
			);
			CLFaults1.4:= Clamp4FB.Faulted AND Clamp_Count>=4; 		(*Interlock Clamp Fault with Clamp Count Configuration Data*)
		(*Clamp5*)
		Clamp5FB(
			(*All sensor input mapping and solenoid mapping is done external to FB by end deployment*)
			Home_Sensor:= MAP_Clamp5_HomeSens,
			Work_Sensor:= MAP_Clamp5_WorkSens,
			Home_Solenoid:= Enable_Motion AND (CMD_Tool_To_HOME OR MAP_Clamp5_HomeReqd),
			Work_Solenoid:= Enable_Motion AND (CMD_Tool_To_WORK OR MAP_Clamp5_WorkReqd),
			Home_Delay:= T#0.1s,
			Work_Delay:= T#0.1s ,
			Fault_Delay:= T#3s ,
			In_Home_Position=> Clamp5HOME,
			In_Work_Position=> Clamp5WORK,
			);
			CLFaults1.5:= Clamp5FB.Faulted AND Clamp_Count>=5; 		(*Interlock Clamp Fault with Clamp Count Configuration Data*)
		(*Clamp6*)
		Clamp6FB(
			(*All sensor input mapping and solenoid mapping is done external to FB by end deployment*)
			Home_Sensor:= MAP_Clamp6_HomeSens,
			Work_Sensor:= MAP_Clamp6_WorkSens,
			Home_Solenoid:= Enable_Motion AND (CMD_Tool_To_HOME OR MAP_Clamp6_HomeReqd),
			Work_Solenoid:= Enable_Motion AND (CMD_Tool_To_WORK OR MAP_Clamp6_WorkReqd),
			Home_Delay:= T#0.1s,
			Work_Delay:= T#0.1s ,
			Fault_Delay:= T#3s ,
			In_Home_Position=> Clamp6HOME,
			In_Work_Position=> Clamp6WORK,
			);
			CLFaults1.6:= Clamp6FB.Faulted AND Clamp_Count>=6; 		(*Interlock Clamp Fault with Clamp Count Configuration Data*)
		(*Clamp7*)
		Clamp7FB(
			(*All sensor input mapping and solenoid mapping is done external to FB by end deployment*)
			Home_Sensor:= MAP_Clamp7_HomeSens,
			Work_Sensor:= MAP_Clamp7_WorkSens,
			Home_Solenoid:= Enable_Motion AND (CMD_Tool_To_HOME OR MAP_Clamp7_HomeReqd),
			Work_Solenoid:= Enable_Motion AND (CMD_Tool_To_WORK OR MAP_Clamp7_WorkReqd),
			Home_Delay:= T#0.1s,
			Work_Delay:= T#0.1s ,
			Fault_Delay:= T#3s ,
			In_Home_Position=> Clamp7HOME,
			In_Work_Position=> Clamp7WORK,
			);
			CLFaults1.7:= Clamp7FB.Faulted AND Clamp_Count>=7; 		(*Interlock Clamp Fault with Clamp Count Configuration Data*)
		(*Clamp8*)
		Clamp8FB(
			(*All sensor input mapping and solenoid mapping is done external to FB by end deployment*)
			Home_Sensor:= MAP_Clamp8_HomeSens,
			Work_Sensor:= MAP_Clamp8_WorkSens,
			Home_Solenoid:= Enable_Motion AND (CMD_Tool_To_HOME OR MAP_Clamp8_HomeReqd),
			Work_Solenoid:= Enable_Motion AND (CMD_Tool_To_WORK OR MAP_Clamp8_WorkReqd),
			Home_Delay:= T#0.1s,
			Work_Delay:= T#0.1s ,
			Fault_Delay:= T#3s ,
			In_Home_Position=> Clamp8HOME,
			In_Work_Position=> Clamp8WORK,
			);
			CLFaults1.8:= Clamp8FB.Faulted AND Clamp_Count>=8; 		(*Interlock Clamp Fault with Clamp Count Configuration Data*)
		(*Clamp9*)
		Clamp9FB(
			(*All sensor input mapping and solenoid mapping is done external to FB by end deployment*)
			Home_Sensor:= MAP_Clamp9_HomeSens,
			Work_Sensor:= MAP_Clamp9_WorkSens,
			Home_Solenoid:= Enable_Motion AND (CMD_Tool_To_HOME OR MAP_Clamp9_HomeReqd),
			Work_Solenoid:= Enable_Motion AND (CMD_Tool_To_WORK OR MAP_Clamp9_WorkReqd),
			Home_Delay:= T#0.1s,
			Work_Delay:= T#0.1s ,
			Fault_Delay:= T#3s ,
			In_Home_Position=> Clamp9HOME,
			In_Work_Position=> Clamp9WORK,
			);
			CLFaults1.9:= Clamp9FB.Faulted AND Clamp_Count>=9; 		(*Interlock Clamp Fault with Clamp Count Configuration Data*)
		(*Clamp10*)
		Clamp10FB(
			(*All sensor input mapping and solenoid mapping is done external to FB by end deployment*)
			Home_Sensor:= MAP_Clamp10_HomeSens,
			Work_Sensor:= MAP_Clamp10_WorkSens,
			Home_Solenoid:= Enable_Motion AND (CMD_Tool_To_HOME OR MAP_Clamp10_HomeReqd),
			Work_Solenoid:= Enable_Motion AND (CMD_Tool_To_WORK OR MAP_Clamp10_WorkReqd),
			Home_Delay:= T#0.1s,
			Work_Delay:= T#0.1s ,
			Fault_Delay:= T#3s ,
			In_Home_Position=> Clamp10HOME,
			In_Work_Position=> Clamp10WORK,
			);
			CLFaults1.10:= Clamp10FB.Faulted AND Clamp_Count>=10; 		(*Interlock Clamp Fault with Clamp Count Configuration Data*)
		(*Clamp11*)
		Clamp11FB(
			(*All sensor input mapping and solenoid mapping is done external to FB by end deployment*)
			Home_Sensor:= MAP_Clamp11_HomeSens,
			Work_Sensor:= MAP_Clamp11_WorkSens,
			Home_Solenoid:= Enable_Motion AND (CMD_Tool_To_HOME OR MAP_Clamp11_HomeReqd),
			Work_Solenoid:= Enable_Motion AND (CMD_Tool_To_WORK OR MAP_Clamp11_WorkReqd),
			Home_Delay:= T#0.1s,
			Work_Delay:= T#0.1s ,
			Fault_Delay:= T#3s ,
			In_Home_Position=> Clamp11HOME,
			In_Work_Position=> Clamp11WORK,
			);
			CLFaults1.11:= Clamp11FB.Faulted AND Clamp_Count>=11; 		(*Interlock Clamp Fault with Clamp Count Configuration Data*)
		(*Clamp12*)
		Clamp12FB(
			(*All sensor input mapping and solenoid mapping is done external to FB by end deployment*)
			Home_Sensor:= MAP_Clamp12_HomeSens,
			Work_Sensor:= MAP_Clamp12_WorkSens,
			Home_Solenoid:= Enable_Motion AND (CMD_Tool_To_HOME OR MAP_Clamp12_HomeReqd),
			Work_Solenoid:= Enable_Motion AND (CMD_Tool_To_WORK OR MAP_Clamp12_WorkReqd),
			Home_Delay:= T#0.1s,
			Work_Delay:= T#0.1s ,
			Fault_Delay:= T#3s ,
			In_Home_Position=> Clamp12HOME,
			In_Work_Position=> Clamp12WORK,
			);
			CLFaults1.12:= Clamp12FB.Faulted AND Clamp_Count>=12; 		(*Interlock Clamp Fault with Clamp Count Configuration Data*)
		(*Clamp13*)
		Clamp13FB(
			(*All sensor input mapping and solenoid mapping is done external to FB by end deployment*)
			Home_Sensor:= MAP_Clamp13_HomeSens,
			Work_Sensor:= MAP_Clamp13_WorkSens,
			Home_Solenoid:= Enable_Motion AND (CMD_Tool_To_HOME OR MAP_Clamp13_HomeReqd),
			Work_Solenoid:= Enable_Motion AND (CMD_Tool_To_WORK OR MAP_Clamp13_WorkReqd),
			Home_Delay:= T#0.1s,
			Work_Delay:= T#0.1s ,
			Fault_Delay:= T#3s ,
			In_Home_Position=> Clamp13HOME,
			In_Work_Position=> Clamp13WORK,
			);
			CLFaults1.13:= Clamp13FB.Faulted AND Clamp_Count>=13; 		(*Interlock Clamp Fault with Clamp Count Configuration Data*)
		(*Clamp14*)
		Clamp14FB(
			(*All sensor input mapping and solenoid mapping is done external to FB by end deployment*)
			Home_Sensor:= MAP_Clamp14_HomeSens,
			Work_Sensor:= MAP_Clamp14_WorkSens,
			Home_Solenoid:= Enable_Motion AND (CMD_Tool_To_HOME OR MAP_Clamp14_HomeReqd),
			Work_Solenoid:= Enable_Motion AND (CMD_Tool_To_WORK OR MAP_Clamp14_WorkReqd),
			Home_Delay:= T#0.1s,
			Work_Delay:= T#0.1s ,
			Fault_Delay:= T#3s ,
			In_Home_Position=> Clamp14HOME,
			In_Work_Position=> Clamp14WORK,
			);
			CLFaults1.14:= Clamp14FB.Faulted AND Clamp_Count>=14; 		(*Interlock Clamp Fault with Clamp Count Configuration Data*)
		(*Clamp15*)
		Clamp15FB(
			(*All sensor input mapping and solenoid mapping is done external to FB by end deployment*)
			Home_Sensor:= MAP_Clamp15_HomeSens,
			Work_Sensor:= MAP_Clamp15_WorkSens,
			Home_Solenoid:= Enable_Motion AND (CMD_Tool_To_HOME OR MAP_Clamp15_HomeReqd),
			Work_Solenoid:= Enable_Motion AND (CMD_Tool_To_WORK OR MAP_Clamp15_WorkReqd),
			Home_Delay:= T#0.1s,
			Work_Delay:= T#0.1s ,
			Fault_Delay:= T#3s ,
			In_Home_Position=> Clamp15HOME,
			In_Work_Position=> Clamp15WORK,
			);
			CLFaults1.15:= Clamp15FB.Faulted AND Clamp_Count>=15; 		(*Interlock Clamp Fault with Clamp Count Configuration Data*)
		(*Clamp16*)
		Clamp16FB(
			(*All sensor input mapping and solenoid mapping is done external to FB by end deployment*)
			Home_Sensor:= MAP_Clamp16_HomeSens,
			Work_Sensor:= MAP_Clamp16_WorkSens,
			Home_Solenoid:= Enable_Motion AND (CMD_Tool_To_HOME OR MAP_Clamp16_HomeReqd),
			Work_Solenoid:= Enable_Motion AND (CMD_Tool_To_WORK OR MAP_Clamp16_WorkReqd),
			Home_Delay:= T#0.1s,
			Work_Delay:= T#0.1s ,
			Fault_Delay:= T#3s ,
			In_Home_Position=> Clamp16HOME,
			In_Work_Position=> Clamp16WORK,
			);
			CLFaults1.16:= Clamp16FB.Faulted AND Clamp_Count>=16; 		(*Interlock Clamp Fault with Clamp Count Configuration Data*)
		(*Clamp17*)
		Clamp17FB(
			(*All sensor input mapping and solenoid mapping is done external to FB by end deployment*)
			Home_Sensor:= MAP_Clamp17_HomeSens,
			Work_Sensor:= MAP_Clamp17_WorkSens,
			Home_Solenoid:= Enable_Motion AND (CMD_Tool_To_HOME OR MAP_Clamp17_HomeReqd),
			Work_Solenoid:= Enable_Motion AND (CMD_Tool_To_WORK OR MAP_Clamp17_WorkReqd),
			Home_Delay:= T#0.1s,
			Work_Delay:= T#0.1s ,
			Fault_Delay:= T#3s ,
			In_Home_Position=> Clamp17HOME,
			In_Work_Position=> Clamp17WORK,
			);
			CLFaults1.17:= Clamp17FB.Faulted AND Clamp_Count>=17; 		(*Interlock Clamp Fault with Clamp Count Configuration Data*)
		(*Clamp18*)
		Clamp18FB(
			(*All sensor input mapping and solenoid mapping is done external to FB by end deployment*)
			Home_Sensor:= MAP_Clamp18_HomeSens,
			Work_Sensor:= MAP_Clamp18_WorkSens,
			Home_Solenoid:= Enable_Motion AND (CMD_Tool_To_HOME OR MAP_Clamp18_HomeReqd),
			Work_Solenoid:= Enable_Motion AND (CMD_Tool_To_WORK OR MAP_Clamp18_WorkReqd),
			Home_Delay:= T#0.1s,
			Work_Delay:= T#0.1s ,
			Fault_Delay:= T#3s ,
			In_Home_Position=> Clamp18HOME,
			In_Work_Position=> Clamp18WORK,
			);
			CLFaults1.18:= Clamp18FB.Faulted AND Clamp_Count>=18; 		(*Interlock Clamp Fault with Clamp Count Configuration Data*)
		(*Clamp19*)
		Clamp19FB(
			(*All sensor input mapping and solenoid mapping is done external to FB by end deployment*)
			Home_Sensor:= MAP_Clamp19_HomeSens,
			Work_Sensor:= MAP_Clamp19_WorkSens,
			Home_Solenoid:= Enable_Motion AND (CMD_Tool_To_HOME OR MAP_Clamp19_HomeReqd),
			Work_Solenoid:= Enable_Motion AND (CMD_Tool_To_WORK OR MAP_Clamp19_WorkReqd),
			Home_Delay:= T#0.1s,
			Work_Delay:= T#0.1s ,
			Fault_Delay:= T#3s ,
			In_Home_Position=> Clamp19HOME,
			In_Work_Position=> Clamp19WORK,
			);
			CLFaults1.19:= Clamp19FB.Faulted AND Clamp_Count>=19; 		(*Interlock Clamp Fault with Clamp Count Configuration Data*)
		(*Clamp20*)
		Clamp20FB(
			(*All sensor input mapping and solenoid mapping is done external to FB by end deployment*)
			Home_Sensor:= MAP_Clamp20_HomeSens,
			Work_Sensor:= MAP_Clamp20_WorkSens,
			Home_Solenoid:= Enable_Motion AND (CMD_Tool_To_HOME OR MAP_Clamp20_HomeReqd),
			Work_Solenoid:= Enable_Motion AND (CMD_Tool_To_WORK OR MAP_Clamp20_WorkReqd),
			Home_Delay:= T#0.1s,
			Work_Delay:= T#0.1s ,
			Fault_Delay:= T#3s ,
			In_Home_Position=> Clamp20HOME,
			In_Work_Position=> Clamp20WORK,
			);
			CLFaults1.20:= Clamp20FB.Faulted AND Clamp_Count>=20; 		(*Interlock Clamp Fault with Clamp Count Configuration Data*)

(*---------------------------------------------------- Group Clamp Sensors ----------------------------------------------------------------*)

	(*Tool All Home*)
	Tool_At_Home.0:= (Clamp1HOME OR Clamp_Count<1)
						AND (Clamp2HOME OR Clamp_Count<2)
						AND (Clamp3HOME OR Clamp_Count<3)
						AND (Clamp4HOME OR Clamp_Count<4)
						AND (Clamp5HOME OR Clamp_Count<5)
						AND (Clamp6HOME OR Clamp_Count<6)
						AND (Clamp7HOME OR Clamp_Count<7)
						AND (Clamp8HOME OR Clamp_Count<8)
						AND (Clamp9HOME OR Clamp_Count<9)
						AND (Clamp10HOME OR Clamp_Count<10)
						AND (Clamp11HOME OR Clamp_Count<11)
						AND (Clamp12HOME OR Clamp_Count<12)
						AND (Clamp13HOME OR Clamp_Count<13)
						AND (Clamp14HOME OR Clamp_Count<14)
						AND (Clamp15HOME OR Clamp_Count<15)
						AND (Clamp16HOME OR Clamp_Count<16)
						AND (Clamp17HOME OR Clamp_Count<17)
						AND (Clamp18HOME OR Clamp_Count<18)
						AND (Clamp19HOME OR Clamp_Count<19)
						AND (Clamp20HOME OR Clamp_Count<20);
	(*Tool All Work*)
	Tool_At_Work.0:= (Clamp1WORK OR Clamp_Count<1)
						AND (Clamp2WORK OR Clamp_Count<2)
						AND (Clamp3WORK OR Clamp_Count<3)
						AND (Clamp4WORK OR Clamp_Count<4)
						AND (Clamp5WORK OR Clamp_Count<5)
						AND (Clamp6WORK OR Clamp_Count<6)
						AND (Clamp7WORK OR Clamp_Count<7)
						AND (Clamp8WORK OR Clamp_Count<8)
						AND (Clamp9WORK OR Clamp_Count<9)
						AND (Clamp10WORK OR Clamp_Count<10)
						AND (Clamp11WORK OR Clamp_Count<11)
						AND (Clamp12WORK OR Clamp_Count<12)
						AND (Clamp13WORK OR Clamp_Count<13)
						AND (Clamp14WORK OR Clamp_Count<14)
						AND (Clamp15WORK OR Clamp_Count<15)
						AND (Clamp16WORK OR Clamp_Count<16)
						AND (Clamp17WORK OR Clamp_Count<17)
						AND (Clamp18WORK OR Clamp_Count<18)
						AND (Clamp19WORK OR Clamp_Count<19)
						AND (Clamp20WORK OR Clamp_Count<20);

(*Note: The remaining Tool_At bits are used for groups and are mapped outside of FB by end deployment*)
	(*Group 1*)
	Tool_At_Home.1:= Tool_At_Home_Grp1;
	Tool_At_Work.1:= Tool_At_Work_Grp1;
	(*Group 2*)
	Tool_At_Home.2:= Tool_At_Home_Grp2;
	Tool_At_Work.2:= Tool_At_Work_Grp2;
	(*Group 3*)
	Tool_At_Home.3:= Tool_At_Home_Grp3;
	Tool_At_Work.3:= Tool_At_Work_Grp3;
	(*Group 4*)
	Tool_At_Home.4:= Tool_At_Home_Grp4;
	Tool_At_Work.4:= Tool_At_Work_Grp4;
	(*Group 5*)
	Tool_At_Home.5:= Tool_At_Home_Grp5;
	Tool_At_Work.5:= Tool_At_Work_Grp5;
	(*Group 6*)
	Tool_At_Home.6:= Tool_At_Home_Grp6;
	Tool_At_Work.6:= Tool_At_Work_Grp6;
	(*Group 7*)
	Tool_At_Home.7:= Tool_At_Home_Grp7;
	Tool_At_Work.7:= Tool_At_Work_Grp7;
	(*Group 8*)
	Tool_At_Home.8:= Tool_At_Home_Grp8;
	Tool_At_Work.8:= Tool_At_Work_Grp8;

(*------------------------------------------------------------ Gather Part Present Sensor Inputs -----------------------------------------------*)
(*Part Present Inputs*)

	(*Part 1 Present*)
		Part_Present1FB(
			(*All Sensor Input mapping and Trigger on/off_1 mapping done external to FB by end deloyment*)
			Sensor_Input:= MAP_PP1_Sens,
			On_Trigger1:= CMD_CheckAllSensors_ON OR MAP_PP1_ReqdOn,
			On_Trigger2:= TRUE,
			Off_Trigger1:= CMD_CheckAllSensors_OFF OR MAP_PP1_ReqdOff,
			On_Trigger2:= TRUE,
			Disable_Faults:= FALSE,
			Fault_Delay:= T#1.5s,
			Status=> Part_Present1,
			);
			PPFaults.1:= Part_Present1FB.Faulted AND Part_Present_Count>=1;		(*Interlock Part Present Fault with Part Present Count Configuration Data*)
	(*Part 2 Present*)
		Part_Present2FB(
			(*All Sensor Input mapping and Trigger on/off_1 mapping done external to FB by end deloyment*)
			Sensor_Input:= MAP_PP2_Sens,
			On_Trigger1:= CMD_CheckAllSensors_ON OR MAP_PP2_ReqdOn,
			On_Trigger2:= TRUE,
			Off_Trigger1:= CMD_CheckAllSensors_OFF OR MAP_PP2_ReqdOff,
			On_Trigger2:= TRUE,
			Disable_Faults:= FALSE,
			Fault_Delay:= T#1.5s,
			Status=> Part_Present2,
			);
			PPFaults.2:= Part_Present2FB.Faulted AND Part_Present_Count>=2;		(*Interlock Part Present Fault with Part Present Count Configuration Data*)
	(*Part 3 Present*)
		Part_Present3FB(
			(*All Sensor Input mapping and Trigger on/off_1 mapping done external to FB by end deloyment*)
			Sensor_Input:= MAP_PP3_Sens,
			On_Trigger1:= CMD_CheckAllSensors_ON OR MAP_PP3_ReqdOn,
			On_Trigger2:= TRUE,
			Off_Trigger1:= CMD_CheckAllSensors_OFF OR MAP_PP3_ReqdOff,
			On_Trigger2:= TRUE,
			Disable_Faults:= FALSE,
			Fault_Delay:= T#1.5s,
			Status=> Part_Present3,
			);
			PPFaults.3:= Part_Present3FB.Faulted AND Part_Present_Count>=3;		(*Interlock Part Present Fault with Part Present Count Configuration Data*)
	(*Part 4 Present*)
		Part_Present4FB(
			(*All Sensor Input mapping and Trigger on/off_1 mapping done external to FB by end deloyment*)
			Sensor_Input:= MAP_PP4_Sens,
			On_Trigger1:= CMD_CheckAllSensors_ON OR MAP_PP4_ReqdOn,
			On_Trigger2:= TRUE,
			Off_Trigger1:= CMD_CheckAllSensors_OFF OR MAP_PP4_ReqdOff,
			On_Trigger2:= TRUE,
			Disable_Faults:= FALSE,
			Fault_Delay:= T#1.5s,
			Status=> Part_Present4,
			);
			PPFaults.4:= Part_Present4FB.Faulted AND Part_Present_Count>=4;		(*Interlock Part Present Fault with Part Present Count Configuration Data*)
	(*Part 5 Present*)
		Part_Present5FB(
			(*All Sensor Input mapping and Trigger on/off_1 mapping done external to FB by end deloyment*)
			Sensor_Input:= MAP_PP5_Sens,
			On_Trigger1:= CMD_CheckAllSensors_ON OR MAP_PP5_ReqdOn,
			On_Trigger2:= TRUE,
			Off_Trigger1:= CMD_CheckAllSensors_OFF OR MAP_PP5_ReqdOff,
			On_Trigger2:= TRUE,
			Disable_Faults:= FALSE,
			Fault_Delay:= T#1.5s,
			Status=> Part_Present5,
			);
			PPFaults.5:= Part_Present5FB.Faulted AND Part_Present_Count>=5;		(*Interlock Part Present Fault with Part Present Count Configuration Data*)
	(*Part 6 Present*)
		Part_Present6FB(
			(*All Sensor Input mapping and Trigger on/off_1 mapping done external to FB by end deloyment*)
			Sensor_Input:= MAP_PP6_Sens,
			On_Trigger1:= CMD_CheckAllSensors_ON OR MAP_PP6_ReqdOn,
			On_Trigger2:= TRUE,
			Off_Trigger1:= CMD_CheckAllSensors_OFF OR MAP_PP6_ReqdOff,
			On_Trigger2:= TRUE,
			Disable_Faults:= FALSE,
			Fault_Delay:= T#1.5s,
			Status=> Part_Present6,
			);
			PPFaults.6:= Part_Present6FB.Faulted AND Part_Present_Count>=6;		(*Interlock Part Present Fault with Part Present Count Configuration Data*)
	(*Part 7 Present*)
		Part_Present7FB(
			(*All Sensor Input mapping and Trigger on/off_1 mapping done external to FB by end deloyment*)
			Sensor_Input:= MAP_PP7_Sens,
			On_Trigger1:= CMD_CheckAllSensors_ON OR MAP_PP7_ReqdOn,
			On_Trigger2:= TRUE,
			Off_Trigger1:= CMD_CheckAllSensors_OFF OR MAP_PP7_ReqdOff,
			On_Trigger2:= TRUE,
			Disable_Faults:= FALSE,
			Fault_Delay:= T#1.5s,
			Status=> Part_Present7,
			);
			PPFaults.7:= Part_Present7FB.Faulted AND Part_Present_Count>=7;		(*Interlock Part Present Fault with Part Present Count Configuration Data*)
	(*Part 8 Present*)
		Part_Present8FB(
			(*All Sensor Input mapping and Trigger on/off_1 mapping done external to FB by end deloyment*)
			Sensor_Input:= MAP_PP8_Sens,
			On_Trigger1:= CMD_CheckAllSensors_ON OR MAP_PP8_ReqdOn,
			On_Trigger2:= TRUE,
			Off_Trigger1:= CMD_CheckAllSensors_OFF OR MAP_PP8_ReqdOff,
			On_Trigger2:= TRUE,
			Disable_Faults:= FALSE,
			Fault_Delay:= T#1.5s,
			Status=> Part_Present8,
			);
			PPFaults.8:= Part_Present8FB.Faulted AND Part_Present_Count>=8;		(*Interlock Part Present Fault with Part Present Count Configuration Data*)

(*---------------------------------------------------- Group Part Present Sensors ----------------------------------------------------------------*)

	(*All Sensors Off*)
	All_Sensors_Off.0:= NOT Part_Present1 AND NOT Part_Present2 AND NOT  Part_Present3
					AND NOT Part_Present4 AND NOT Part_Present5 AND NOT Part_Present6
					AND NOT Part_Present7 AND NOT Part_Present8;
	(*All Sensors On*)
	All_Sensors_On.0:= ((Part_Present1 OR Part_Present_Count<1)
						AND (Part_Present2 OR Part_Present_Count<2)
						AND (Part_Present3 OR Part_Present_Count<3)
						AND (Part_Present4 OR Part_Present_Count<4)
						AND (Part_Present5 OR Part_Present_Count<5)
						AND (Part_Present6 OR Part_Present_Count<6)
						AND (Part_Present7 OR Part_Present_Count<7)
						AND (Part_Present8 OR Part_Present_Count<8))
					OR (All_Sensors_Off.0 AND Dry_Cycle);

(*Note: The remaining All_Sensors_On bits are used for groups and are mapped outside of FB by end deployment*)

	(*All Sensors On Designated for Group 1*)
	All_Sensors_On.1:= (All_Sensors_On_Grp1 AND NOT Dry_Cycle)
					OR (All_Sensors_Off.0 AND Dry_Cycle);
	(*All Sensors Off Designated for Group 1*)
	All_Sensors_Off.1:= All_Sensors_Off_Grp1;

	(*All Sensors On Designated for Group 2*)
	All_Sensors_On.2:= (All_Sensors_On_Grp2 AND NOT Dry_Cycle)
					OR (All_Sensors_Off.0 AND Dry_Cycle);
	(*All Sensors Off Designated for Group 1*)
	All_Sensors_Off.2:= All_Sensors_Off_Grp2;

	(*All Sensors On Designated for Group 3*)
	All_Sensors_On.3:= (All_Sensors_On_Grp3 AND NOT Dry_Cycle)
					OR (All_Sensors_Off.0 AND Dry_Cycle);
	(*All Sensors Off Designated for Group 1*)
	All_Sensors_Off.3:= All_Sensors_Off_Grp3;

	(*All Sensors On Designated for Group 4*)
	All_Sensors_On.4:= (All_Sensors_On_Grp4 AND NOT Dry_Cycle)
					OR (All_Sensors_Off.0 AND Dry_Cycle);
	(*All Sensors Off Designated for Group 1*)
	All_Sensors_Off.4:= All_Sensors_Off_Grp4;

	(*All Sensors On Designated for Group 5*)
	All_Sensors_On.5:= (All_Sensors_On_Grp5 AND NOT Dry_Cycle)
					OR (All_Sensors_Off.0 AND Dry_Cycle);
	(*All Sensors Off Designated for Group 1*)
	All_Sensors_Off.5:= All_Sensors_Off_Grp5;

	(*All Sensors On Designated for Group 6*)
	All_Sensors_On.6:= (All_Sensors_On_Grp6 AND NOT Dry_Cycle)
					OR (All_Sensors_Off.0 AND Dry_Cycle);
	(*All Sensors Off Designated for Group 1*)
	All_Sensors_Off.6:= All_Sensors_Off_Grp6;

	(*All Sensors On Designated for Group 7*)
	All_Sensors_On.7:= (All_Sensors_On_Grp7 AND NOT Dry_Cycle)
					OR (All_Sensors_Off.0 AND Dry_Cycle);
	(*All Sensors Off Designated for Group 1*)
	All_Sensors_Off.7:= All_Sensors_Off_Grp7;

	(*All Sensors On Designated for Group 8*)
	All_Sensors_On.8:= (All_Sensors_On_Grp8 AND NOT Dry_Cycle)
					OR (All_Sensors_Off.0 AND Dry_Cycle);
	(*All Sensors Off Designated for Group 1*)
	All_Sensors_Off.8:= All_Sensors_Off_Grp8;



(*$$$$$$$$$$$$$$$$$$$$$$$$$$$$$$$$$$$$$$$$$$$$$$$$$$$ Faults $$$$$$$$$$$$$$$$$$$$$$$$$$$$$$$$$$$$$$$$$$$$$$$$$$$$$$$*)
	(*Clamp/Cylinder Faults*)
		IF CLFaults1>0
			THEN CLFaulted.1:=TRUE;
		ELSE
			CLFaulted.1:=FALSE;
		END_IF;
	(*Spare Fault Word*)
		IF CLFaults2>0
			THEN CLFaulted.2:=TRUE;
		ELSE
			CLFaulted.2:=FALSE;
		END_IF;
	(*Spare Fault Word*)
		IF CLFaults3>0
			THEN CLFaulted.3:=TRUE;
		ELSE
			CLFaulted.3:=FALSE;
		END_IF;
	(*Spare Fault Word*)
		IF CLFaults4>0
			THEN CLFaulted.4:=TRUE;
		ELSE
			CLFaulted.4:=FALSE;
		END_IF;
	(*Bit 0 is designated as ANY Clamp Fault Word Faulted*)
	IF CLFaulted.1 OR CLFaulted.2 OR CLFaulted.3
		THEN CLFaulted.0:= TRUE;
	ELSE CLFaulted.0 := FALSE;
	END_IF;

	(*Part Present Sensor Faults*)
		IF PPFaults>0
			THEN PPFaulted.0:=TRUE;
		ELSE
			PPFaulted.0:=FALSE;
		END_IF;



(*$$$$$$$$$$$$$$$$$$$$$$$$$$$$$$$$$$$$$$$$$$$$$$ Transfer Standard Outputs $$$$$$$$$$$$$$$$$$$$$$$$$$$$$$$$$$$$$$$$$$$*)
	(*Transfer General Status and I/O Images for Display On HMI*)
	Discrete_Image.CLFaults1:= CLFaults1;
	Discrete_Image.CLFaults2:= CLFaults2;
	Discrete_Image.CLFaults3:= CLFaults3;
	Discrete_Image.CLFaults4:= CLFaults4;
	Discrete_Image.CLFaulted:= CLFaulted;
	Discrete_Image.PPFaults:= PPFaults;
	Discrete_Image.PPFaulted:= PPFaulted;

	Discrete_Image.N01:=N01;
	Discrete_Image.N02:=N02;
	Discrete_Image.N03:=N03;
	Discrete_Image.N04:=N04;
	Discrete_Image.N05:=N05;
	Discrete_Image.N06:=N06;
	Discrete_Image.N07:=N07;
	Discrete_Image.N08:=N08;
	Discrete_Image.N09:=N09;
	Discrete_Image.N100:=N100;
	Discrete_Image.N100_STAT:=N100_STAT;

	Discrete_Image.ECatSlave_Cable_Breaks:= ECatSlave_Cable_Breaks;
	Discrete_Image.Input_Node_Count:= Input_Node_Count;
	Discrete_Image.VB_Node_Count:= VB_Node_Count;

(*---------------------------------------------------------------------------------------- Transfer ACKS Back to external of FB ----------------------------------------------------------*)

	ACK_AllSensors_OFF:= CMD_CheckAllSensors_OFF AND All_Sensors_Off.0;
	ACK_AllSensors_ON:= CMD_CheckAllSensors_ON AND All_Sensors_On.0;

	ACK_SensorsOFF_Grp1:= CMD_CheckSensorsOFF_Grp1 AND All_Sensors_Off.1;
	ACK_SensorsON_Grp1:= CMD_CheckSensorsON_Grp1 AND All_Sensors_On.1;
	ACK_SensorsOFF_Grp2:= CMD_CheckSensorsOFF_Grp2 AND All_Sensors_Off.2;
	ACK_SensorsON_Grp2:= CMD_CheckSensorsON_Grp2 AND All_Sensors_On.2;
	ACK_SensorsOFF_Grp3:= CMD_CheckSensorsOFF_Grp3 AND All_Sensors_Off.3;
	ACK_SensorsON_Grp3:= CMD_CheckSensorsON_Grp3 AND All_Sensors_On.3;
	ACK_SensorsOFF_Grp4:= CMD_CheckSensorsOFF_Grp4 AND All_Sensors_Off.4;
	ACK_SensorsON_Grp4:= CMD_CheckSensorsON_Grp4 AND All_Sensors_On.4;
	ACK_SensorsOFF_Grp5:= CMD_CheckSensorsOFF_Grp5 AND All_Sensors_Off.5;
	ACK_SensorsON_Grp5:= CMD_CheckSensorsON_Grp5 AND All_Sensors_On.5;
	ACK_SensorsOFF_Grp6:= CMD_CheckSensorsOFF_Grp6 AND All_Sensors_Off.6;
	ACK_SensorsON_Grp6:= CMD_CheckSensorsON_Grp6 AND All_Sensors_On.6;
	ACK_SensorsOFF_Grp7:= CMD_CheckSensorsOFF_Grp7 AND All_Sensors_Off.7;
	ACK_SensorsON_Grp7:= CMD_CheckSensorsON_Grp7 AND All_Sensors_On.7;
	ACK_SensorsOFF_Grp8:= CMD_CheckSensorsOFF_Grp8 AND All_Sensors_Off.8;
	ACK_SensorsON_Grp8:= CMD_CheckSensorsON_Grp8 AND All_Sensors_On.8;

	IF LH_Part_In_EOAT_Grp AND NOT LH_EOAT_Empty_Grp
		THEN LH_Part_In_EOAT:= TRUE;
	ELSIF  LH_EOAT_Empty_Grp
		THEN LH_Part_In_EOAT:= FALSE;
	END_IF;

	IF RH_Part_In_EOAT_Grp AND NOT RH_EOAT_Empty_Grp
		THEN RH_Part_In_EOAT:= TRUE;
	ELSIF  RH_EOAT_Empty_Grp
		THEN RH_Part_In_EOAT:= FALSE;
	END_IF;

	IF (LH_Part_In_EOAT_Grp AND RH_Part_In_EOAT_Grp)
		AND (NOT LH_EOAT_Empty_Grp AND NOT RH_EOAT_Empty_Grp)
		THEN Part_In_EOAT:= TRUE;
	ELSIF  (LH_EOAT_Empty_Grp AND RH_EOAT_Empty_Grp)
		THEN Part_In_EOAT:= FALSE;
	END_IF;

	ACK_Tool_At_WORK:= CMD_Tool_To_WORK AND Tool_At_WORK.0;
	ACK_Tool_At_HOME:= CMD_Tool_To_HOME AND Tool_At_HOME.0;

	ACK_ClampsAtWORK_Grp1:= CMD_ClampsToWORK_Grp1 AND Tool_At_WORK.1;
	ACK_ClampsAtHOME_Grp1:= CMD_ClampsToHOME_Grp1 AND Tool_At_HOME.1;
	ACK_ClampsAtWORK_Grp2:= CMD_ClampsToWORK_Grp2 AND Tool_At_WORK.2;
	ACK_ClampsAtHOME_Grp2:= CMD_ClampsToHOME_Grp2 AND Tool_At_HOME.2;
	ACK_ClampsAtWORK_Grp3:= CMD_ClampsToWORK_Grp3 AND Tool_At_WORK.3;
	ACK_ClampsAtHOME_Grp3:= CMD_ClampsToHOME_Grp3 AND Tool_At_HOME.3;
	ACK_ClampsAtWORK_Grp4:= CMD_ClampsToWORK_Grp4 AND Tool_At_WORK.4;
	ACK_ClampsAtHOME_Grp4:= CMD_ClampsToHOME_Grp4 AND Tool_At_HOME.4;
	ACK_ClampsAtWORK_Grp5:= CMD_ClampsToWORK_Grp5 AND Tool_At_WORK.5;
	ACK_ClampsAtHOME_Grp5:= CMD_ClampsToHOME_Grp5 AND Tool_At_HOME.5;
	ACK_ClampsAtWORK_Grp6:= CMD_ClampsToWORK_Grp6 AND Tool_At_WORK.6;
	ACK_ClampsAtHOME_Grp6:= CMD_ClampsToHOME_Grp6 AND Tool_At_HOME.6;
	ACK_ClampsAtWORK_Grp7:= CMD_ClampsToWORK_Grp7 AND Tool_At_WORK.7;
	ACK_ClampsAtHOME_Grp7:= CMD_ClampsToHOME_Grp7 AND Tool_At_HOME.7;
	ACK_ClampsAtWORK_Grp8:= CMD_ClampsToWORK_Grp8 AND Tool_At_WORK.8;
	ACK_ClampsAtHOME_Grp8:= CMD_ClampsToHOME_Grp8 AND Tool_At_HOME.8;


(*-----------------------------------------------------------------------------------------Transfer Valve Outputs --------------------------------------------------------------------------------*)

	(*Valve 1, A+B*)
	(*Clamp Group 1*)
		Valve1FB
			(
			Enable_Motion:= Enable_Motion ,
			Enable_Latch:= FALSE,					(*Enabling Runs Valve as detent type (maintained solenoids*)
			Enable_SideA_PreCharge:= FALSE,		(*Enabling Turns Side A PreCharge Active, reset when Side B is energized in Auto*)
			Enable_SideB_PreCharge:= FALSE,		(*Enabling Turns Side B PreCharge Active, reset when Side A is energized in Auto*)
			PreCharge_Time:= T#0.1S,
			Enable_Auto_Commands:= Enable_Motion,
			In_Auto_SideA_Command:= CMD_Tool_To_WORK OR CMD_ClampsToWORK_Grp1,
			In_Auto_SideB_Command:= CMD_Tool_To_HOME OR CMD_ClampsToHOME_Grp1,
			Enable_Manual_Commands:= FALSE,
			In_Manual_SideA_Command:= FALSE,
			In_Manual_SideB_Command:= FALSE,
			SideA_Indicator:= Tool_At_WORK.1,
			SideB_Indicator:= Tool_At_HOME.1,
			TurnOn_SideA_SOL=> N100.Q.0,
			TurnOn_SideB_SOL=> N100.Q.1,
			TurnOn_SideA_Indicator=> ,
			TurnOn_SideB_Indicator=>
			 );
	(*Valve 2, A+B*)
	(*Clamp Group 2*)
		Valve2FB
			(
			Enable_Motion:= Enable_Motion ,
			Enable_Latch:= FALSE,					(*Enabling Runs Valve as detent type (maintained solenoids*)
			Enable_SideA_PreCharge:= FALSE,		(*Enabling Turns Side A PreCharge Active, reset when Side B is energized in Auto*)
			Enable_SideB_PreCharge:= FALSE,		(*Enabling Turns Side B PreCharge Active, reset when Side A is energized in Auto*)
			PreCharge_Time:= T#0.1S,
			Enable_Auto_Commands:= Enable_Motion,
			In_Auto_SideA_Command:= CMD_ClampsToWORK_Grp2,
			In_Auto_SideB_Command:= CMD_ClampsToHome_Grp2,
			Enable_Manual_Commands:= FALSE,
			In_Manual_SideA_Command:= FALSE,
			In_Manual_SideB_Command:= FALSE,
			SideA_Indicator:= Tool_At_WORK.2,
			SideB_Indicator:= Tool_At_HOME.2,
			TurnOn_SideA_SOL=> N100.Q.2,
			TurnOn_SideB_SOL=> N100.Q.3,
			TurnOn_SideA_Indicator=> ,
			TurnOn_SideB_Indicator=>
			 );
	(*Valve 3, A+B*)
	(*Clamp Group 3*)
		Valve3FB
			(
			Enable_Motion:= Enable_Motion ,
			Enable_Latch:= FALSE,					(*Enabling Runs Valve as detent type (maintained solenoids*)
			Enable_SideA_PreCharge:= FALSE,		(*Enabling Turns Side A PreCharge Active, reset when Side B is energized in Auto*)
			Enable_SideB_PreCharge:= FALSE,		(*Enabling Turns Side B PreCharge Active, reset when Side A is energized in Auto*)
			PreCharge_Time:= T#0.1S,
			Enable_Auto_Commands:= Enable_Motion,
			In_Auto_SideA_Command:= CMD_ClampsToWORK_Grp3,
			In_Auto_SideB_Command:= CMD_ClampsToHome_Grp3,
			Enable_Manual_Commands:= FALSE,
			In_Manual_SideA_Command:= FALSE,
			In_Manual_SideB_Command:= FALSE,
			SideA_Indicator:= Tool_At_WORK.3,
			SideB_Indicator:= Tool_At_HOME.3,
			TurnOn_SideA_SOL=> N100.Q.4,
			TurnOn_SideB_SOL=> N100.Q.5,
			TurnOn_SideA_Indicator=> ,
			TurnOn_SideB_Indicator=>
			 );
	(*Valve 4, A+B*)
	(*Clamp Group 4*)
		Valve4FB
			(
			Enable_Motion:= Enable_Motion ,
			Enable_Latch:= FALSE,					(*Enabling Runs Valve as detent type (maintained solenoids*)
			Enable_SideA_PreCharge:= FALSE,		(*Enabling Turns Side A PreCharge Active, reset when Side B is energized in Auto*)
			Enable_SideB_PreCharge:= FALSE,		(*Enabling Turns Side B PreCharge Active, reset when Side A is energized in Auto*)
			PreCharge_Time:= T#0.1S,
			Enable_Auto_Commands:= Enable_Motion,
			In_Auto_SideA_Command:= CMD_ClampsToWORK_Grp4,
			In_Auto_SideB_Command:= CMD_ClampsToHome_Grp4,
			Enable_Manual_Commands:= FALSE,
			In_Manual_SideA_Command:= FALSE,
			In_Manual_SideB_Command:= FALSE,
			SideA_Indicator:= Tool_At_WORK.4,
			SideB_Indicator:= Tool_At_HOME.4,
			TurnOn_SideA_SOL=> N100.Q.6,
			TurnOn_SideB_SOL=> N100.Q.7,
			TurnOn_SideA_Indicator=> ,
			TurnOn_SideB_Indicator=>
			 );
	(*Valve 5, A+B*)
	(*Clamp Group 5*)
		Valve5FB
			(
			Enable_Motion:= Enable_Motion ,
			Enable_Latch:= FALSE,					(*Enabling Runs Valve as detent type (maintained solenoids*)
			Enable_SideA_PreCharge:= FALSE,		(*Enabling Turns Side A PreCharge Active, reset when Side B is energized in Auto*)
			Enable_SideB_PreCharge:= FALSE,		(*Enabling Turns Side B PreCharge Active, reset when Side A is energized in Auto*)
			PreCharge_Time:= T#0.1S,
			Enable_Auto_Commands:= Enable_Motion,
			In_Auto_SideA_Command:= CMD_ClampsToWORK_Grp5,
			In_Auto_SideB_Command:= CMD_ClampsToHome_Grp5,
			Enable_Manual_Commands:= FALSE,
			In_Manual_SideA_Command:= FALSE,
			In_Manual_SideB_Command:= FALSE,
			SideA_Indicator:= Tool_At_WORK.5,
			SideB_Indicator:= Tool_At_HOME.5,
			TurnOn_SideA_SOL=> N100.Q.8,
			TurnOn_SideB_SOL=> N100.Q.9,
			TurnOn_SideA_Indicator=> ,
			TurnOn_SideB_Indicator=>
			 );
	(*Valve 6, A+B*)
	(*Clamp Group 6*)
		Valve6FB
			(
			Enable_Motion:= Enable_Motion ,
			Enable_Latch:= FALSE,					(*Enabling Runs Valve as detent type (maintained solenoids*)
			Enable_SideA_PreCharge:= FALSE,		(*Enabling Turns Side A PreCharge Active, reset when Side B is energized in Auto*)
			Enable_SideB_PreCharge:= FALSE,		(*Enabling Turns Side B PreCharge Active, reset when Side A is energized in Auto*)
			PreCharge_Time:= T#0.1S,
			Enable_Auto_Commands:= Enable_Motion,
			In_Auto_SideA_Command:= CMD_ClampsToWORK_Grp6,
			In_Auto_SideB_Command:= CMD_ClampsToHome_Grp6,
			Enable_Manual_Commands:= FALSE,
			In_Manual_SideA_Command:= FALSE,
			In_Manual_SideB_Command:= FALSE,
			SideA_Indicator:= Tool_At_WORK.6,
			SideB_Indicator:= Tool_At_HOME.6,
			TurnOn_SideA_SOL=> N100.Q.10,
			TurnOn_SideB_SOL=> N100.Q.11,
			TurnOn_SideA_Indicator=> ,
			TurnOn_SideB_Indicator=>
			 );
	(*Valve 7, A+B*)
	(*Clamp Group 7*)
		Valve7FB
			(
			Enable_Motion:= Enable_Motion ,
			Enable_Latch:= FALSE,					(*Enabling Runs Valve as detent type (maintained solenoids*)
			Enable_SideA_PreCharge:= FALSE,		(*Enabling Turns Side A PreCharge Active, reset when Side B is energized in Auto*)
			Enable_SideB_PreCharge:= FALSE,		(*Enabling Turns Side B PreCharge Active, reset when Side A is energized in Auto*)
			PreCharge_Time:= T#0.1S,
			Enable_Auto_Commands:= Enable_Motion,
			In_Auto_SideA_Command:= CMD_ClampsToWORK_Grp7,
			In_Auto_SideB_Command:= CMD_ClampsToHome_Grp7,
			Enable_Manual_Commands:= FALSE,
			In_Manual_SideA_Command:= FALSE,
			In_Manual_SideB_Command:= FALSE,
			SideA_Indicator:= Tool_At_WORK.7,
			SideB_Indicator:= Tool_At_HOME.7,
			TurnOn_SideA_SOL=> N100.Q.12,
			TurnOn_SideB_SOL=> N100.Q.13,
			TurnOn_SideA_Indicator=> ,
			TurnOn_SideB_Indicator=>
			 );
	(*Valve 8, A+B*)
	(*Clamp Group 8*)
		Valve8FB
			(
			Enable_Motion:= Enable_Motion ,
			Enable_Latch:= FALSE,					(*Enabling Runs Valve as detent type (maintained solenoids*)
			Enable_SideA_PreCharge:= FALSE,		(*Enabling Turns Side A PreCharge Active, reset when Side B is energized in Auto*)
			Enable_SideB_PreCharge:= FALSE,		(*Enabling Turns Side B PreCharge Active, reset when Side A is energized in Auto*)
			PreCharge_Time:= T#0.1S,
			Enable_Auto_Commands:= Enable_Motion,
			In_Auto_SideA_Command:= CMD_ClampsToWORK_Grp8,
			In_Auto_SideB_Command:= CMD_ClampsToHome_Grp8,
			Enable_Manual_Commands:= FALSE,
			In_Manual_SideA_Command:= FALSE,
			In_Manual_SideB_Command:= FALSE,
			SideA_Indicator:= Tool_At_WORK.8,
			SideB_Indicator:= Tool_At_HOME.8,
			TurnOn_SideA_SOL=> N100.Q.14,
			TurnOn_SideB_SOL=> N100.Q.15,
			TurnOn_SideA_Indicator=> ,
			TurnOn_SideB_Indicator=>
			 );

END_FUNCTION_BLOCK

// ---- POUs/FBs/FB_GTAC_Motoman_20170531.TcPOU
(*FB for use with Motoman XRC, NX100 and DX100 Series Robot Controller
	Equiped with HMS AnyBus Profibus Card, Maped as 32 Byte I/O Size:

	Author(s): Brent Lekx-Toniolo/Rob Remillard of Sodecia GTAC.; 
	Version 1.0: August 2012
		- Initial Concept
------------------------------------------------------------------------------------------
REVISION NOTES:
	 Version 20121204
		Changes from v1 include:
			- Changed to Generic HW Images and Added Type Conversion Calls
			- Increased Profibus Image Sizes from 32 bytes I/O to 64 bytes I/O		
			- Added variables for more functionality
			- Change to Naming Convention to include date as version
	 Version 20130405
			- General De-bug During first commisioning of this FB
	Version 20141016
			- Small updates for Weld Contoller Fault Abstraction: b.lekx-toniolo
	Version 20150103
			- changed FB_In declaration. RR/JVD
	Version 20150120:
	- Updated Generic FBIN Instance, b.lekx-toniolo
	Version 20150128:
	- Added code for "teach Interlock" status message, b.lekx-toniolo
	Version 20150819:
	- Changed 4 uses of INT_TO_BYTE conversion types to UINT_TO_BYTE to avoid compiler warnings messages, b.lekx-toniolo
	Version 20151105:
	- Changed from profibus to EtherCAT, b.lekx-toniolo
	Version 20170531:
	- Updates for Options, b.lekx-toniolo


------------------------------------------------------------------------------------------

*)

FUNCTION_BLOCK FB_GTAC_Motoman_20170531
	VAR_INPUT
		Enable_FB: BOOL;
		FB_In: udt_Generic_Robot_FBIN_CUSTOM; (*Inputs to FB*)

	END_VAR

	VAR
(*Hardware Data Types*)
		(*Develop Discrete Node*)
		T01 AT %I*: udt_EK1100;				(*Ecat Bus Coupler*)
		T02_STAT AT %I*: udt_EL6900_STAT_20160426;	(*EL Safety CPU*)
		T02_CMD AT %Q*: udt_EL6900_CMD_20121204;
		T03 AT %I*: udt_EL1904_v2;				(*EL Safety Inputs*)
		T04 AT %I*: udt_EL1904_v2;				(*EL Safety Inputs*)
		T05 AT %I*: udt_EL1904_v2;				(*EL Safety Inputs*)
		T06 AT %I*: udt_EL1904_v2;				(*EL Safety Inputs*)
		T07 AT %I*: udt_EL1904_v2;				(*EL Safety Inputs*)
		T08 AT %I*: udt_EL2904RO_v2;			(*EL Safety Outputs, Set to "I" as this terminal is safety rated, therefore read only!*)
		T09 AT %I*: udt_EL2904RO_v2; 			(*EL Safety Outputs, Set to "I" as this terminal is safety rated, therefore read only!*)
		T10 AT %I*: udt_EL2904RO_v2; 			(*EL Safety Outputs, Set to "I" as this terminal is safety rated, therefore read only!*)

		(*Develop Profibus Node*)
		In_From_HW AT %I*: udt_GenericRobot_AnyFieldbus_InputBytes_20220421;
		In_From_ECAT: udt_EtherCAT_Motoman_Input_20151105;

		Out_To_HW AT %Q*: udt_GenericRobot_AnyFieldbus_OutputBytes_20220421;
		Out_To_ECAT: udt_EtherCAT_Motoman_Output_20151105;

(* Nodes States*)
		DiscreteNode_OK: BOOL;
		ECATNode_OK: BOOL;
(*Cable Connection Warning Flags*)
		EK1100_NotPresent :BOOL;			(*Coupler is Not Present on Bus when expected*)
		EK1100_PortC_MissingLink: BOOL;      (*Port C of EK1100 is OUT*)
(*Safety Internals*)
		PendEstop_Ok: BOOL;		(*Robot Teach Pendant Estop Button OK, See Rxx Print Package, Page P03*)
		ContEstop_Ok: BOOL;		(*Robot Controller Estop Estop Button OK, See Rxx Print Package, Page P03*)

		ZoneClear_Detect_On: BOOL; (*Hardware Detects that Robot is Clear of All Human Interf Zones*)
		ZoneClear_Detect_Off: BOOL; (*Hardware Detects that Robot may not be Clear of All Human Interf Zones*)

		Estop_Relays_On: BOOL;		(*Robot Estop Relays Are On, See Rxx Print Package, Page P05 and P08 *)
		Estop_Relays_Off: BOOL;		(*Robot Estop Relays Are Off*)
		SafetyGate_Relays_On: BOOL;	(*Robot Safety Gate Relays Are On, See Rxx Print Package, Page P05 and P08*)
		SafetyGate_Relays_Off: BOOL;	(*Robot Safety Gate Relays Are Off*)
		EOAT_Relays_On: BOOL;		(*Robot EOAT Relays Are On, See Rxx Print Package, Page P05 and P09*)
		EOAT_Relays_Off: BOOL;		(*Robot EOAT Relays Are Off*)

		Table_SideA_At_Robots: BOOL;		(*Side A of Turntable at Robots (Ext Axis S1)*)
		Table_SideB_At_Robots: BOOL;		(*Side B of Turntable at Robots (Ext Axis S1)*)

		Zone1_Detected_Clear: BOOL; (*Hardware Detects that Robot is Clear of Human Interf#1*)
		Zone1_Detected_NotClear: BOOL; (*Hardware Detects that Robot is In Human Interf#1*)
		Zone2_Detected_Clear: BOOL; (*Hardware Detects that Robot is Clear of Human Interf#2*)
		Zone2_Detected_NotClear: BOOL; (*Hardware Detects that Robot is In Human Interf#2*)
		Zone3_Detected_Clear: BOOL; (*Hardware Detects that Robot is Clear of Human Interf#3*)
		Zone3_Detected_NotClear: BOOL; (*Hardware Detects that Robot is In Human Interf#3*)
		Zone4_Detected_Clear: BOOL; (*Hardware Detects that Robot is Clear of Human Interf#4*)
		Zone4_Detected_NotClear: BOOL; (*Hardware Detects that Robot is In Human Interf#4*)
		Zone5_Detected_Clear: BOOL; (*Hardware Detects that Robot is Clear of Human Interf#5*)
		Zone5_Detected_NotClear: BOOL; (*Hardware Detects that Robot is In Human Interf#5*)
		Zone6_Detected_Clear: BOOL; (*Hardware Detects that Robot is Clear of Human Interf#6*)
		Zone6_Detected_NotClear: BOOL; (*Hardware Detects that Robot is In Human Interf#6*)
		Zone7_Detected_Clear: BOOL; (*Hardware Detects that Robot is Clear of Human Interf#7*)
		Zone7_Detected_NotClear: BOOL; (*Hardware Detects that Robot is In Human Interf#7*)
		Zone8_Detected_Clear: BOOL; (*Hardware Detects that Robot is Clear of Human Interf#8*)
		Zone8_Detected_NotClear: BOOL; (*Hardware Detects that Robot is In Human Interf#8*)


(*Standard Internals*)
		(*System Inputs*)
		Operating: BOOL;
		Servos_Are_On: BOOL;
		S1_Servo_On: BOOL; (*Externa Axis S1 Servo On DX100_3_MIG*)
		S2_Servo_On: BOOL; (*Externa Axis S2 Servo On DX100_3_MIG*)
		S3_Servo_On: BOOL; (*Externa Axis S3 Servo On DX100_3_MIG*)
		Top_Of_Master: BOOL;
		Faulted: BOOL;
		Battery_Alarm: BOOL;
		In_Remote: BOOL;
		In_Play: BOOL;
		In_Teach: BOOL;
		In_Cube1: BOOL;
		In_Cube2: BOOL;
		In_Cube24: BOOL;	(* Work Home for XRC2001*)
		In_Cube32: BOOL; (*Work Home for NX100*)
		In_Cube64: BOOL;	(*Work Home for DX100*)
		R1_In_Cube64: BOOL; (*Work Home for R1 for DX100_3_MIG*)
		R2_In_Cube63: BOOL; (*Work Home for R2 for DX100_3_MIG*)
		R3_In_Cube62: BOOL; (*Work Home for R3 for DX100_3_MIG*)
		All_At_Home: BOOL; (*All 3 Robots At Work Home*)
		Intermediate_Start_OK: BOOL;
		Any_Rob_ArcAlarm: BOOL; (*Any of 3 Robots Arc Alarm*)
		Any_Rob_WireStick: BOOL; (*Any of 3 Robots Wire Sticking*)
		In_Cube3: BOOL;
		In_Cube4: BOOL;
		In_Cube5: BOOL;
		In_Cube10: BOOL;
		Collision_Detect_Valid: BOOL;
		Holding: BOOL;

		(*Standard Inputs*)
		(*From OG5*)
		WCU1_StepperNearMax_1: BOOL;
		WCU1_StepperAtMax_1: BOOL;
		WCU1_StepperNearMax_2: BOOL;
		WCU1_StepperAtMax_2: BOOL;
		WCU2_StepperNearMax_1: BOOL;
		WCU2_StepperAtMax_1: BOOL;
		WCU2_StepperNearMax_2: BOOL;
		WCU2_StepperAtMax_2: BOOL;
		Master_Job_Req_ExtAxisOn: BOOL;
		(*Weld Controller Common*)
		Weld_Controller_Faulted: BOOL;

		(*From OG6*)
		Clear_Of_EquipInterf1: BOOL;
		Clear_Of_EquipInterf2: BOOL;
		Clear_Of_EquipInterf3: BOOL;
		Clear_Of_EquipInterf4: BOOL;
		Clear_Of_EquipInterf5: BOOL;
		Clear_Of_EquipInterf6: BOOL;
		Clear_Of_EquipInterf7: BOOL;
		Clear_Of_EquipInterf8: BOOL;
		(*From OG7*)
		Clear_Of_HumanInterf1: BOOL;
		Clear_Of_HumanInterf2: BOOL;
		Clear_Of_HumanInterf3: BOOL;
		Clear_Of_HumanInterf4: BOOL;
		Clear_Of_HumanInterf5: BOOL;
		Clear_Of_HumanInterf6: BOOL;
		Clear_Of_HumanInterf7: BOOL;
		Clear_Of_HumanInterf8: BOOL;
		(*From OG8*)
		Fix_ID_Ack: UINT;
		(*From OG9*)
		EOAT_ID_Ack: UINT;
		(*From OG10*)
		Model_ID_Ack: UINT;
		(*From OG11*)
		Task_ID_Ack: UINT;
		(*From OG12*)
		Peripheral_Req: UINT;
		(*From OG13*)
		At_Pounce: BOOL;
		LHPart_In_EOAT: BOOL;
		RHPart_In_EOAT: BOOL;
		Clear_To_Unclamp: BOOL;
		Task_Completed: BOOL;
		(*From OG14*)
		Clear_Of_RobotInterfs: UINT;
		(*From OG17*)
		EOAT_Req:UINT;
		(*From OG#26*)
		WCU1_NoFaults: BOOL;
		(*From OG#30*)
		WCU2_NoFaults: BOOL;


(*Internal Code Variables*)
		Location_Index: UINT;			(*The So Called Location Index is used to Mux and emux Information to and From the Robot Based on its Working Location*)
		At_Home: BOOL;				(*Robot is At Work Or Intermediate Home*)
		R1_At_Home: BOOL;			(*Robot 1 at home in triple robot controller DX100_3_MIG*)
		R2_At_Home: BOOL;			(*Robot 2 at home in triple robot controller DX100_3_MIG*)
		R3_At_Home: BOOL;			(*Robot 3 at home in triple robot controller DX100_3_MIG*)
		At_EquipInterf1: BOOL;
		At_EquipInterf2: BOOL;
		At_EquipInterf3: BOOL;
		At_EquipInterf4: BOOL;
		At_EquipInterf5: BOOL;
		At_EquipInterf6: BOOL;
		At_EquipInterf7: BOOL;
		At_EquipInterf8: BOOL;

		At_HumanInterf1: BOOL;
		At_HumanInterf2: BOOL;
		At_HumanInterf3: BOOL;
		At_HumanInterf4: BOOL;
		At_HumanInterf5: BOOL;
		At_HumanInterf6: BOOL;
		At_HumanInterf7: BOOL;
		At_HumanInterf8: BOOL;

		(*InterfsOK*)
		OK_At_EquipInterf1: BOOL;
		OK_At_EquipInterf2: BOOL;
		OK_At_EquipInterf3: BOOL;
		OK_At_EquipInterf4: BOOL;
		OK_At_EquipInterf5: BOOL;
		OK_At_EquipInterf6: BOOL;
		OK_At_EquipInterf7: BOOL;
		OK_At_EquipInterf8: BOOL;
		OK_At_EquipInterfALL: BOOL;

		OK_At_HumanInterf1: BOOL;
		OK_At_HumanInterf2: BOOL;
		OK_At_HumanInterf3: BOOL;
		OK_At_HumanInterf4: BOOL;
		OK_At_HumanInterf5: BOOL;
		OK_At_HumanInterf6: BOOL;
		OK_At_HumanInterf7: BOOL;
		OK_At_HumanInterf8: BOOL;
		OK_At_HumanInterfALL: BOOL;

		OK_At_RobotInterfs: UINT;
		OK_At_RobotInterfsALL: BOOL;

		Ready: BOOL;					(* Robot is Ready*)
		ID_Acks_OK: BOOL;				(*Robot has Ack'd proper Task and Fix ID*)
		All_Interfs_Ok: BOOL;				(*All Interferences with Human and Equipment Zones OK*)
		Servos_Req: BOOL;				(*Request to Turn On Servos*)
		Servos_Req_Delay: TON;			(*Delay Servos On Request*)
		Servos_Off_Req: BOOL;				(*Request to Turn Servos OFF*)
		Play_Delay: TON; 					(*NX100 Only*)
		Start_Robot_Scan: BOOL;			(*Start Robot*)
		Hold_Robot: BOOL;				(*Hold Robot*)
		Fix_ID_FLT: BOOL;
		EOAT_ID_FLT: BOOL;
		Model_ID_FLT: BOOL;
		Task_ID_FLT: BOOL;
		Ack_ID_FLT: BOOL;
		Ack_ID_TMR: TON;
		Comp_Ack_TMR: TON;
		Stay_Off: BOOL:=FALSE;			(*Local Always Off*)
		Motoman_Types:					(*Enumeration of Robot Types*)
		(
			ERC:=1,
			MRC:=2,
			XRC:=10,
			NX100:=20,
			DX100:=30,
			DX100_Dual:=31,
			DX100_3_MIG:=41
		);
		Robot_Is_AutoRestart: BOOL;		(*Robot Is Auto Restart Type, for Internal Robots etc*)
	Temp1: BOOL;
	Temp2: BOOL;
	Temp3: BOOL;
	Temp4: BOOL;
	Temp5: BOOL;
	Temp6: BOOL;
	Temp7: BOOL;
	Temp8: BOOL;

	END_VAR
	VAR PERSISTENT
		(*Place data variables here that must be retained during power outage*)
	END_VAR

	VAR_OUTPUT
		FB_Ok: BOOL;
		Status: INT;
		Input_Image: udt_GenericRobot_AnyFieldbus_InputBytes_20220421;
		Output_Image: udt_GenericRobot_AnyFieldbus_OutputBytes_20220421;
		Discrete_Image: udt_RobotDiscreteNode_ImageSSCCv46_20131001;

	END_VAR

	(*Check Robot Type and set FB_OK to True if range is ok*)
	IF FB_In.Robot_Type>0 AND FB_In.Robot_Type<50
		THEN
		FB_OK:= TRUE;
	ELSE
		FB_OK:= FALSE;
	END_IF;
(*----------------- First Gather an Input Image in Generic Byte Type and convert TO Kuka Specific Type*)

In_From_ECAT:= FUN_GTAC_GenericRobotInputImage_TO_MOTOMAN32(In_From_HW);

(*$$$$$$$$$$$$$$$$$$$$$$$$$$$$$$$$$$$$$$$$$$$$$$$$Gather Status Of Hardware $$$$$$$$$$$$$$$$$$$$$$$$$$$$$$$$$$$$$$$$$$$$$$$$$$$$*)
	(*Discrete I/O Node (Node On Robot Controller Door)*)
	IF T01.InfoData.State=8 AND T02_Stat.InfoData.State=8 AND T03.InfoData.State=8 AND T04.InfoData.State=8 AND T05.InfoData.State=8
		AND T06.InfoData.State=8 AND T07.InfoData.State=8 AND T08.InfoData.State=8 AND T09.InfoData.State=8
		 AND T10.InfoData.State=8
		THEN DiscreteNode_OK:=TRUE;
	ELSE DiscreteNode_OK:=FALSE;
	END_IF;
	(*Ethercat Node (Anybus PCI card)*)
	IF In_From_ECAT.InfoData.State=8
		THEN ECATNode_OK:=TRUE;
	ELSE ECATNode_OK:=FALSE;
	END_IF;

(*Develop Port Connection Warning Flags*)
	IF T01.InfoData.State=257 (*State Machine for Slave Not Present*)
		THEN EK1100_NotPresent:= TRUE;
	ELSE EK1100_NotPresent := FALSE;
	END_IF;

	IF T01.InfoData.State=17416 (*State Machine for Link Missing at Port C*)
		THEN EK1100_PortC_MissingLink:= TRUE; (*PortC is OUT Port*)
	ELSE EK1100_PortC_MissingLink := FALSE;
	END_IF;
(*$$$$$$$$$$$$$$$$$$$$$$$$$$$$$$$$$$$$$$$$$$$$$$$$$$ Gather All Safety I/O $$$$$$$$$$$$$$$$$$$$$$$$$$$$$$$$$$$$$$$$$$$$$$$$$$$$$$$$$$$$$*)
	PendEstop_OK:=T03.I.0 AND T03.I.1;
	ContEstop_OK:=T03.I.2 AND T03.I.3;

	ZoneClear_Detect_On:= T04.I.2 AND T04.I.3;
	ZoneClear_Detect_Off:= NOT ZoneClear_Detect_On;

	Estop_Relays_On:= NOT T05.I.0;
	Estop_Relays_Off:= T05.I.0;
	SafetyGate_Relays_On:= NOT T05.I.1;
	SafetyGate_Relays_Off:= T05.I.1;
	EOAT_Relays_On:= NOT T05.I.2;
	EOAT_Relays_Off:= T05.I.2;

	Table_SideA_At_Robots:= T06.I.0 AND T06.I.1;				(*Turntable External axis S1*)
	Table_SideB_At_Robots:= T06.I.2 AND T06.I.3;				(*Turntable External axis S1*)

	Zone1_Detected_Clear:= T06.I.0 AND T06.I.1;
	Zone1_Detected_NotClear:= NOT Zone1_Detected_Clear;
	Zone2_Detected_Clear:= T06.I.2 AND T06.I.3;
	Zone2_Detected_NotClear:= NOT Zone2_Detected_Clear;
	Zone3_Detected_Clear:= T07.I.0 AND T07.I.1;
	Zone3_Detected_NotClear:= NOT Zone3_Detected_Clear;
	Zone4_Detected_Clear:= T07.I.2 AND T07.I.3;
	Zone4_Detected_NotClear:= NOT Zone4_Detected_Clear;
	Zone5_Detected_Clear:= TRUE;
	Zone5_Detected_NotClear:= NOT Zone5_Detected_Clear;
	Zone6_Detected_Clear:= TRUE;
	Zone6_Detected_NotClear:= NOT Zone6_Detected_Clear;
	Zone7_Detected_Clear:= TRUE;
	Zone7_Detected_NotClear:= NOT Zone7_Detected_Clear;
	Zone8_Detected_Clear:= TRUE;
	Zone8_Detected_NotClear:= NOT Zone8_Detected_Clear;


(*$$$$$$$$$$$$$$$$$$$$$$$$$$$$$$$$$$$$$$$$$$$$$$$$$$$$Gather All Standard I/O $$$$$$$$$$$$$$$$$$$$$$$$$$$$$$$$$$$$$$$$$$$$$$$$$$$$$$$$$$$$$*)
	Operating:= In_From_ECAT.SYS.0;								(*Operating*)
	Servos_Are_On:= In_From_ECAT.SYS.1;							(*Servo Power On*)
	Top_Of_Master:= In_From_ECAT.SYS.2;							(*Top Of Master*)
	Faulted:= In_From_ECAT.SYS.3;									(*Faulted*)
	Battery_Alarm:= In_From_ECAT.SYS.4;							(*Battery Alarm*)
	In_Remote:= In_From_ECAT.SYS.5;								(*In Remote*)
	In_Play:= In_From_ECAT.SYS.6;									(*In Play*)
	In_Teach:= In_From_ECAT.SYS.7;								(*In Teach*)
	In_Cube1:= In_From_ECAT.SYS.8;								(*In Cube 1*)
	IF FB_In.Robot_Type=DX100_3_MIG
		THEN
			In_Cube10:= In_From_ECAT.SYS.9;						(*R2 In Cube 10*)
	END_IF;
	(*XRC Home*)
	IF FB_In.Robot_Type=XRC
		THEN In_Cube24:= In_From_ECAT.SYS.10;					(*In Home XRC*)
	END_IF;
	(*NX100*)
	IF FB_In.Robot_Type=NX100
		THEN In_Cube32:= In_From_ECAT.SYS.10;					(*In Home NX100*)
	END_IF;
	(*DX100 Single and Dual and Triple Mig*)
	IF FB_In.Robot_Type=DX100
		THEN In_Cube64:= In_From_ECAT.SYS.10;					(*In Home DX100*)
	ELSIF FB_In.Robot_Type=DX100_Dual
		THEN In_Cube64:= In_From_ECAT.SYS.10;					(*In Home DX100*)
	ELSIF FB_In.Robot_Type=DX100_3_MIG
		THEN All_At_Home:= In_From_ECAT.SYS.10;					(*All 3 Robots At Home DX100_3_MIG*)
	END_IF;

	Intermediate_Start_OK:= In_From_ECAT.SYS.11;					(*Intermediate Start OK*)

	IF (FB_In.Robot_Type=XRC) OR (FB_In.Robot_Type=NX100)
		OR (FB_In.Robot_Type=DX100) OR (FB_In.Robot_Type=DX100_Dual)
		THEN In_Cube3:= In_From_ECAT.SYS.12;						(*In Cube 3*)
	ELSIF FB_In.Robot_Type=DX100_3_MIG
		THEN Collision_Detect_Valid:= In_From_ECAT.SYS.12;			(*Collision Detect Valid*)
	END_IF;

	IF (FB_In.Robot_Type=XRC) OR (FB_In.Robot_Type=NX100)
		OR (FB_In.Robot_Type=DX100) OR (FB_In.Robot_Type=DX100_Dual)
		THEN In_Cube4:= In_From_ECAT.SYS.13;						(*In Cube 4*)
	ELSIF FB_In.Robot_Type=DX100_3_MIG
		THEN Any_Rob_ArcAlarm:= In_From_ECAT.SYS.13;			(*Arc Alarm*)
	END_IF;

	IF (FB_In.Robot_Type=XRC) OR (FB_In.Robot_Type=NX100)
		OR (FB_In.Robot_Type=DX100) OR (FB_In.Robot_Type=DX100_Dual)
		THEN Collision_Detect_Valid:= In_From_ECAT.SYS.14;			(*Collision Detect Valid*)
	ELSIF FB_In.Robot_Type=DX100_3_MIG
		THEN Any_Rob_WireStick:= In_From_ECAT.SYS.14;			(*Any of 3 Robots Wire Sticking*)
	END_IF;

	IF (FB_In.Robot_Type=XRC) OR (FB_In.Robot_Type=NX100)
		OR (FB_In.Robot_Type=DX100) OR (FB_In.Robot_Type=DX100_Dual)
		THEN
			Holding:= In_From_ECAT.SYS.15;						(*Holding*)
	ELSE
			In_Cube5:= In_From_ECAT.SYS.15;						(*R3 In Cube 5*)
	END_IF;

	(*OG#4*)
	R1_In_Cube64:= In_From_ECAT.OG4.0;							(*R1 In Cube 64 DX100_3_MIG*)
	R2_In_Cube63:= In_From_ECAT.OG4.1;							(*R2 In Cube 63 DX100_3_MIG*)
	R3_In_Cube62:= In_From_ECAT.OG4.2;							(*R3 In Cube 62 DX100_3_MIG*)

	IF FB_In.Robot_Type=DX100_Dual
		THEN
		WCU1_StepperNearMax_1:= In_From_ECAT.OG4.6;				(*WCU1 Stepper Near Max 1*)
		WCU1_StepperAtMax_1:= In_From_ECAT.OG4.7;				(*WCU1 Stepper At Max 1*)
	ELSIF FB_In.Robot_Type=DX100_3_MIG
		THEN
		Holding:= In_From_ECAT.OG4.7;								(*Holding DX100_3_MIG*)
	END_IF;

	(*OG#5*)
	S1_Servo_On:= In_From_ECAT.OG5.0;							(*External Axis S1 Servo On DX100_3_MIG*)
	S2_Servo_On:= In_From_ECAT.OG5.1;							(*External Axis S2 Servo On DX100_3_MIG*)
	S3_Servo_On:= In_From_ECAT.OG5.2;							(*External Axis S3 Servo On DX100_3_MIG*)
	Master_Job_Req_ExtAxisOn:= In_From_ECAT.OG5.2;				(*Master Job Request for External Axis Servo On*)

	IF FB_In.Robot_Type=DX100_Dual
		THEN
		WCU2_StepperNearMax_1:= In_From_ECAT.OG5.6;				(*WCU2 Stepper Near Max 1*)
		WCU2_StepperAtMax_1:= In_From_ECAT.OG5.7;				(*WCU2 Stepper At Max 1*)
	END_IF;

	IF FB_In.Robot_Type<>DX100_Dual
		THEN
		WCU1_StepperNearMax_1:= In_From_ECAT.OG5.6;				(*WCU1 Stepper Near MAX 1*)
		WCU1_StepperAtMax_1:= In_From_ECAT.OG5.7;				(*WCU1 Stepper At Max 1*)
	END_IF;

	(*OG#6*)
	Clear_Of_EquipInterf1:= In_From_ECAT.OG6.0 ;
	Clear_Of_EquipInterf2:= In_From_ECAT.OG6.1;
	Clear_Of_EquipInterf3:= In_From_ECAT.OG6.2;
	Clear_Of_EquipInterf4:= In_From_ECAT.OG6.3;
	Clear_Of_EquipInterf5:= In_From_ECAT.OG6.4 ;
	Clear_Of_EquipInterf6:= In_From_ECAT.OG6.5;
	Clear_Of_EquipInterf7:= In_From_ECAT.OG6.6;
	Clear_Of_EquipInterf8:= In_From_ECAT.OG6.7;
	(*OG#7*)
	Clear_Of_HumanInterf1:= In_From_ECAT.OG7.0 ;
	Clear_Of_HumanInterf2:= In_From_ECAT.OG7.1;
	Clear_Of_HumanInterf3:= In_From_ECAT.OG7.2 ;
	Clear_Of_HumanInterf4:= In_From_ECAT.OG7.3 ;
	Clear_Of_HumanInterf5:= In_From_ECAT.OG7.4;
	Clear_Of_HumanInterf6:= In_From_ECAT.OG7.5 ;
	Clear_Of_HumanInterf7:= In_From_ECAT.OG7.6 ;
	Clear_Of_HumanInterf8:= In_From_ECAT.OG7.7;
	(*OG#8*)
	EOAT_ID_Ack:=In_From_ECAT.OG8;
	(*OG#9*)
	Fix_ID_Ack:=In_From_ECAT.OG9;
	(*OG#10*)
	Model_ID_Ack:= In_From_ECAT.OG10;
	(*OG#11*)
	Task_ID_Ack:=In_From_ECAT.OG11;
	(*OG#12*)
	Peripheral_Req.0:= In_From_ECAT.OG12.0;
	Peripheral_Req.1:= In_From_ECAT.OG12.1;
	Peripheral_Req.2:= In_From_ECAT.OG12.2;
	Peripheral_Req.3:= In_From_ECAT.OG12.3;
	Peripheral_Req.4:= In_From_ECAT.OG12.4;
	Peripheral_Req.5:= In_From_ECAT.OG12.5;
	Peripheral_Req.6:= In_From_ECAT.OG12.6;
	Peripheral_Req.7:= In_From_ECAT.OG12.7;
	(*OG#13*)
	At_Pounce:= In_From_ECAT.OG13.0;
	LHPart_IN_EOAT:= In_From_ECAT.OG13.1;
	RHPart_In_EOAT:= In_From_ECAT.OG13.2;
	Clear_To_Unclamp:= In_From_ECAT.OG13.3;
	(*Delay Complete*)
	Task_Completed:= In_From_ECAT.OG13.7 AND At_Home;
	(*OG#14*)
	Clear_Of_RobotInterfs.0:= In_From_ECAT.OG14.0;
	Clear_Of_RobotInterfs.1:= In_From_ECAT.OG14.1;
	Clear_Of_RobotInterfs.2:= In_From_ECAT.OG14.2;
	Clear_Of_RobotInterfs.3:= In_From_ECAT.OG14.3;
	Clear_Of_RobotInterfs.4:= In_From_ECAT.OG14.4;
	Clear_Of_RobotInterfs.5:= In_From_ECAT.OG14.5;
	Clear_Of_RobotInterfs.6:= In_From_ECAT.OG14.6;
	Clear_Of_RobotInterfs.7:= In_From_ECAT.OG14.7;
	(*OG#17*)
	EOAT_Req.0:= In_From_ECAT.OG17.0;
	EOAT_Req.1:= In_From_ECAT.OG17.1;
	EOAT_Req.2:= In_From_ECAT.OG17.2;
	EOAT_Req.3:= In_From_ECAT.OG17.3;
	EOAT_Req.4:= In_From_ECAT.OG17.4;
	EOAT_Req.5:= In_From_ECAT.OG17.5;
	EOAT_Req.6:= In_From_ECAT.OG17.6;
	EOAT_Req.7:= In_From_ECAT.OG17.7;

	(*DEBUG, the folowing section must be checked onsight!!!!! - contact b.lekx-toniolo, 16-Oct-2014*)
	(*!!!!!!!!!!!!!!!!!!!!!!!!!!!!!!!!!!!!!!!!!!!!*)
	(*OG#26*)
	WCU1_NoFaults:= In_From_ECAT.OG26.1;
	(*OG#30*)
	WCU2_NoFaults:= In_From_ECAT.OG30.1;

	(*Gather WCU Information, take into account number of WCUs robot is interfaced to*)
		IF FB_In.Options.WeldCont_Amount = 1
			THEN Weld_Controller_Faulted:= NOT WCU1_NoFaults;
		ELSIF FB_In.Options.WeldCont_Amount = 2
			THEN Weld_Controller_Faulted:= NOT WCU1_NoFaults OR NOT WCU2_NoFaults;
		ELSE Weld_Controller_Faulted:= FALSE;
		END_IF;
	(*!!!!!!!!!!!!!!!!!!!!!!!!!!!!!!!!!!!!!!!!!!!!*)

(*$$$$$$$$$$$$$$$$$$$$$$$$$$$$$$$$$$$$$$$$$$$$$$$$$$ Internal Code $$$$$$$$$$$$$$$$$$$$$$$$$$$$$$$$$$$$$$$$$$$$$$$$$$$$$$$$*)
	(*Develop Location Index Number Based On Which Interference Location to Robot Is Working In*)
	IF FALSE
		THEN Location_Index:=0;
	ELSIF At_HumanInterf1
		THEN Location_Index:=1;
	ELSIF At_HumanInterf2
		THEN Location_Index:=2;
	ELSIF At_HumanInterf3
		THEN Location_Index:=3;
	ELSIF At_HumanInterf4
		THEN Location_Index:=4;
	ELSIF At_HumanInterf5
		THEN Location_Index:=5;
	ELSIF At_HumanInterf6
		THEN Location_Index:=6;
	ELSIF At_HumanInterf7
		THEN Location_Index:=7;
	ELSIF At_HumanInterf8
		THEN Location_Index:=8;
	ELSIF At_EquipInterf1
		THEN Location_Index:=9;
	ELSIF At_EquipInterf2
		THEN Location_Index:=10;
	ELSIF At_EquipInterf3
		THEN Location_Index:=11;
	ELSIF At_EquipInterf4
		THEN Location_Index:=12;
	ELSIF At_EquipInterf5
		THEN Location_Index:=13;
	ELSIF At_EquipInterf6
		THEN Location_Index:=14;
	ELSIF At_EquipInterf7
		THEN Location_Index:=15;
	ELSIF At_EquipInterf8
		THEN Location_Index:=16;
	ELSE
		Location_Index:=0;
	END_IF;

	(*Place Limits on Location Index as it will be used to access Arrays (Prevent Out of Bounds)*)
	IF Location_Index>16
		THEN Location_Index:=16;
	ELSIF Location_Index<0
		THEN Location_Index:=0;
	END_IF;

